// POUs/Functions/Pumps/FB_PTM_TurboDrive
(* This Function block provides basic turbo control for Leybold Turbo Drive 300, Turbo Drive 400 *)
(* TD20 Classic Via Remote X1 Connector 9-way PLC interface*)
FUNCTION_BLOCK FB_PTM_TurboDrive
VAR_IN_OUT
	
END_VAR
VAR_INPUT
	i_xExtILKOk : BOOL; // Connect to external interlock logic, TRUE if not used.
END_VAR
VAR_OUTPUT
{attribute 'pytmc' := '
    pv: 
	'}
	iq_stPtm	:	ST_LeyboldPTM;
END_VAR
VAR
	xRunOk	:	BOOL;
	tofRemoteDelay	:	TOF;
	
	
	(*IO*)
	i_xAtSpd AT%I*: BOOL; // Normaml operation when true
	i_xFaultNC AT%I*: BOOL; // Error Active when no Error is present
	q_RunDO AT%Q*: BOOL; // Start/Stop

END_VAR

(* Basic Turbo Control *)
(* This Function block provides basic turbo control for Leybold Turbo Drive 300, Turbo Drive 400 *)
(* TD20 Classic Via Remote X1 Connector 9-way PLC interface*)
(* M. Ghaly Jan. 2019 *)

(* Interlock Sum *)
iq_stPtm.xExtRunOk:= i_xExtILKOk;
xRunOk := iq_stPtm.xExtRunOk AND iq_stPtm.i_xNCError;

(* Basic pump supervisory section *)
IF xRunOk THEN
	iq_stPtm.q_RunDO := iq_stPTM.xRunSW;
ELSE
	iq_stPtm.xRunSW:=FALSE;
	iq_stPtm.q_RunDO:=FALSE;
END_IF

(*Pump States*)
IF (iq_stPtm.i_xFault) THEN
		iq_stPtm.eState := pumpFAULT;
		iq_stPtm.xRunSW:=FALSE;
		iq_stPtm.q_RunDO:=FALSE;
	ELSIF (iq_stPtm.q_RunDO) AND (iq_stPtm.i_xAtSpd) THEN
		iq_stPtm.eState := pumpRUNNING;
	ELSIF (iq_stPtm.q_RunDO) AND NOT (iq_stPtm.i_xAtSpd) THEN
		iq_stPtm.eState := pumpSTARTING; 
	ELSIF NOT (iq_stPtm.q_RunDO) THEN
		iq_stPtm.eState := pumpSTOPPED; 	
END_IF;
			

(*I/O soft mapping*)
ACT_IO();

ACTION ACT_IO:
(*Inputs*)
iq_stPtm.i_xAtSpd := i_xAtSpd;
iq_stPtm.i_xNCError := i_xFaultNC;
iq_stPtm.i_xFault := NOT i_xFaultNC;



(*Outputs*)
q_RunDO := iq_stPtm.q_RunDO;
END_ACTION

METHOD PUBLIC M_Run : BOOL
VAR_INPUT
	run:bool; // set to true to run, false to stop;
END_VAR

this^.iq_stPtm.xRunSW := run;
END_METHOD

END_FUNCTION_BLOCK

// POUs/Functions/Pumps/FB_PTM_TwisTorr
(* This function block does basic controls FOR the Agilent TwisTorr 304 FS with on board Controller.
 Turns off pump in the event of errors/ warnings. Provides interlocking interface.*)
FUNCTION_BLOCK FB_PTM_TwisTorr
VAR_INPUT
	i_xExtILKOk : BOOL; // Connect to external interlock logic, TRUE if not used.
	
END_VAR
VAR_OUTPUT
	{attribute 'pytmc' := ' pv: '}
	iq_stPtm	:	ST_PTM;
END_VAR
VAR
	xRunOk	:	BOOL;
	(*IO*)
	i_xAtSpd AT%I*: BOOL; // Normaml operation when true
	i_xFault AT%I*: BOOL; // Error // this open collector output signal is ON when a system fault condition is detected

	q_RunDO AT%Q*: BOOL; // Start/Stop

END_VAR


(* Interlock Sum *)
iq_stPtm.xExtRunOk:= i_xExtILKOk;
xRunOk := iq_stPtm.xExtRunOk AND NOT iq_stPtm.i_xFault;

(* Basic pump supervisory section *)
IF xRunOk THEN
	iq_stPtm.q_RunDO := iq_stPTM.xRunSW;
ELSE
	iq_stPtm.xRunSW:=FALSE;
	iq_stPtm.q_RunDO:=FALSE;
END_IF

(*Pump STATE*)
IF iq_stPtm.i_xFault THEN 
	iq_stPtm.eState := pumpFAULT;
ELSIF NOT iq_stPtm.q_RunDO AND NOT iq_stPTM.i_xFault THEN
	iq_stPtm.eState := pumpSTOPPED;
ELSIF NOT iq_stPtm.i_xAtSpd  AND iq_stPtm.q_RunDO THEN
	iq_stPtm.eState := pumpSTARTING;
ELSIF iq_stPtm.i_xAtSpd AND iq_stPtm.q_RunDO THEN
	iq_stPtm.eState := pumpRUNNING;
ELSE 
	iq_stPtm.eState := pumpFAULT;
END_IF

(*I/O soft mapping*)
ACT_IO();

ACTION ACT_IO:
(*Inputs*)
iq_stPtm.i_xAtSpd := i_xAtSpd;
iq_stPtm.i_xFault := i_xFault;


(*Outputs*)
q_RunDO := iq_stPtm.q_RunDO;
END_ACTION

METHOD PUBLIC M_Run : BOOL
VAR_INPUT
	run:bool; // set to true to run, false to stop;
END_VAR

this^.iq_stPtm.xRunSW := run;
END_METHOD

END_FUNCTION_BLOCK

// POUs/Functions/Pumps/FB_ScrollPump
(* This Function block provides basic  control for Scroll Pumps *)
(* Turn on scroll pump if the Turbo Vent Valve is closed. *)
(* Cannot turn off scroll pump if turb is running. delay scroll off 150s.*)  

FUNCTION_BLOCK FB_ScrollPump
VAR_IN_OUT

END_VAR
VAR_OUTPUT
	{attribute 'pytmc' := '
    pv:
	'}
	iq_stPFO	:	ST_RoughPump;
END_VAR
VAR_INPUT
	TurboIsON : BOOL;
	xExtIlk : BOOL;
END_VAR
VAR
	Tmr_TOF : TOF;
	tTimerDuration : Time:= T#150S;
	//Previous_RunSW : BOOL;
	// Digital Output to be linked
	q_xRunDo AT%Q*	:   BOOL; 
END_VAR

//Turn on scroll pump if the Turbo Vent Valve is closed. So you are not just
// pumping air and accomplishing nothing

// cannot turn off scroll pump if turb is running. delay scroll off 150s.  
iq_stPFO.xIlkOK := xExtIlk;// and NOT Tmr_TOF.Q;

Tmr_TOF(IN:=TurboIsON, PT := tTimerDuration);

IF iq_stPFO.xIlkOK THEN
	iq_stPFO.q_xRunDo := (Tmr_TOF.Q OR iq_stPFO.pv_xRunSW);
ELSE
	iq_stPFO.q_xRunDo := FALSE;
END_IF

iq_stPFO.pv_xRunSW := iq_stPFO.q_xRunDo;

(*State evaluation*)
IF NOT iq_stPFO.q_xRunDo THEN
	iq_stPFO.eState := pumpSTOPPED;	
ELSE
	iq_stPFO.eState := pumpRUNNING;
END_IF

(*soft io Mapping*)
IO();

ACTION IO:
q_xRunDo:= iq_stPFO.q_xRunDo;
END_ACTION

METHOD PUBLIC M_Run : BOOL
VAR_INPUT
	run:bool; // set to true to run, false to stop;
END_VAR

this^.iq_stPFO.pv_xRunSW := run;
END_METHOD

END_FUNCTION_BLOCK

// POUs/Functions/Valves/functions/F_RoughPumpInlet_ILK
(*
	Determine whether a pump attached to the inlet of a roughing pump is safe to open. 
	
	Return true, signaling it is safe to open when the roughing pump is confirmed to be working. 
*)

FUNCTION F_RoughPumpInlet_ILK : BOOL
VAR_INPUT
	ScrollPump	:	ST_RoughPump;
END_VAR
VAR
END_VAR


F_RoughPumpInlet_ILK := (ScrollPump.eState = pumpRUNNING); (* Confirm that the roughing pump is running before opening the valve *)

END_FUNCTION

// POUs/Functions/Valves/functions/F_TURBO_VRC_ILK
(* Close the vic if the roughing pump pirani loses its at-vac setpoint while the turbo is pumping *)
FUNCTION F_TURBO_VRC_ILK : BOOL
VAR_INPUT

	i_xHiVac 	: BOOL;
	i_xRunPTM	: BOOL;
	i_xFLVac	: BOOL;

END_VAR
VAR

	rHysterisis : REAL := 0;

	xInterlock: BOOL;
	rTolerance: REAL := 20;
END_VAR

(* Close the vic if the roughing pump pirani loses its at-vac setpoint while the turbo is pumping *)
F_TURBO_VRC_ILK := (NOT i_xHiVac AND NOT i_xRunPTM AND NOT i_xFLVac) OR
					(NOT i_xRunPTM AND i_xFLVac) OR
					(i_xRunPTM AND i_xFLVac);

END_FUNCTION

// POUs/Functions/Valves/functions/F_TurboGateValve_ILK
(* This Function Block evaluates the ILK condition of the Turbo Gate valve *)
(* The logic Protects the Turbo pump from inlet pressure above the SP*)

FUNCTION F_TurboGateValve_ILK : BOOL (* function return TRUE when ILK is OK*)
VAR_INPUT
	i_Turbo : ST_PTM; // Turbo Pump
	i_stISG : ST_VG; //Gauge measuring inlet Pressure e.g Pirani
END_VAR
VAR
END_VAR

(* This Function Block evaluates the ILK condition of the Turbo Gate valve *)
(* The logic Protects the Turbo pump from inlet pressure above the SP*)
F_TurboGateValve_ILK := (NOT (i_Turbo.eState = pumpSTOPPED) AND NOT (i_Turbo.eState = pumpFAULT))
						AND (i_stISG.xPRESS_OK AND i_stISG.rPRESS < i_Turbo.rInletPressureSP);

END_FUNCTION

// POUs/Functions/Valves/functions/F_TurboGateValve_Protection_ILK
(* This Function Block evaluates the ILK condition of the Turbo Gate valve *)
(* The logic Protects the Turbo pump from inlet pressure above the SP*)
(* And Protects the Turbo pump from backing pressure above the SP*)
(* And Protects the Turbo pump in the case of backing pump not running*)

FUNCTION F_TurboGateValve_Protection_ILK : BOOL (* function return TRUE when ILK is OK*)
VAR_INPUT
	i_Turbo : ST_PTM; // Turbo Pump
	i_stISG : ST_VG; //Gauge measuring inlet Pressure e.g Pirani
	i_stBSG : ST_VG; //Gauge measuring backing Pressure e.g Pirani
	ScrollPump	:	ST_RoughPump; // Roughing pump
END_VAR
VAR
END_VAR

(* This Function Block evaluates the ILK condition of the Turbo Gate valve *)
(* The logic Protects the Turbo pump from inlet pressure above the SP*)
F_TurboGateValve_Protection_ILK := (NOT (i_Turbo.eState = pumpSTOPPED) AND NOT (i_Turbo.eState = pumpFAULT))
						AND (i_stISG.xPRESS_OK AND i_stISG.rPRESS < i_Turbo.rInletPressureSP)
						AND (i_stBSG.xPRESS_OK AND i_stBSG.rPRESS < i_Turbo.rBackingPressureSP)
						AND (ScrollPump.eState = pumpRUNNING);

END_FUNCTION

// POUs/Functions/Valves/functions/F_VALVE_REL_ILK
(* OK, this is going to be a general-use function that will return whether the ratio of the pressures given is less than x orders of magnitude.
True iff 10^(-x) < a/b < 10^x.  Simple, right?  Just make sure it gets a positive order of magnitude and the pressures aren't 0. ~Scott *)   

FUNCTION F_VALVE_REL_ILK : BOOL
VAR_INPUT
	i_stUSG	:	ST_VG; // Upstream Gague
	i_stDSG	:	ST_VG; // Downstream Gague
	//Orders of magnitude allowed between up/downstream pressures for valve to open. Must be real positive integer.
	i_iOrdersMagnitude: INT;
END_VAR
VAR
	rPressRatio : REAL;
	rMaxRatioAllowed	:	LREAL := EXPT(10,i_iOrdersMagnitude);
	rMinRatioAllowed	:	LREAL := EXPT(10,(-i_iOrdersMagnitude));
END_VAR

(* S. Stubbs 11/2015 *)

(* OK, this is going to be a general-use function that will return whether the ratio of the pressures given is less than x orders of magnitude.
True iff 10^(-x) < a/b < 10^x.  Simple, right?  Just make sure it gets a positive order of magnitude and the pressures aren't 0. ~Scott *)   

(* Find ratio *)

IF i_stDSG.rPRESS <> 0 THEN
	rPressRatio := i_stUSG.rPRESS / i_stDSG.rPRESS;

	F_VALVE_REL_ILK := rPressRatio < rMaxRatioAllowed AND rMinRatioAllowed < rPressRatio;
ELSE
	F_VALVE_REL_ILK := FALSE;
END_IF

END_FUNCTION

// POUs/Functions/Valves/functions/F_VRC_DIODE_ILK
(* The principle is simple, a VRC should never open when B side pressure is greater than 
the A side pressure. *)

FUNCTION F_VRC_DIODE_ILK : BOOL
VAR_INPUT

	i_stPGA : ST_VG; // A side pressure gauge
	i_stPGB	: ST_VG; // B side pressure gauge

END_VAR
VAR

	rHysterisis : REAL := 0;

	xInterlock: BOOL;
	rTolerance: REAL := 20;
END_VAR

(* The principle is simple, a VRC should never open when B side pressure is greater than the A side pressure. *)
rTolerance := 20;
F_VRC_DIODE_ILK := ((i_stPGA.rPRESS + rTolerance >= i_stPGB.rPRESS + rHysterisis) OR i_stPGA.xBAKEOUT) AND i_stPGA.xPRESS_OK AND i_stPGB.xPRESS_OK;

(* OK it gets a bit more complicated with hysterisis,

Now, if the F_VIC_DIODE_ILK is FALSE then some hysterisis is added to the B side. But if it's OK then we just stick with making sure that the A side is greater than the B side

*)
(*
IF NOT F_VIC_DIODE_ILK THEN
Hysterisis := 40;
ELSE
Hysterisis := 0;
END_IF
*)

END_FUNCTION

// POUs/Functions/Valves/Interfaces/FB_TVGC_ADS
(* This function block is created for interface devices between different PLC*)
(* Not all the fields in the original structure is required, just few signals *)
(*Use with FB_ADS_WATCHDOG on remotePLC*)
FUNCTION_BLOCK FB_TVGC_ADS
VAR_INPUT
	sNetId : String; //NetID of the Destination PLC controller
	nPort : int; // port number
	sVarName : string;// the variable name of the (device) declared function block.
	iWatchdog:UDINT;//The watchdog variable name written to by the remote plc
END_VAR
VAR_OUTPUT
	{attribute 'pytmc' := 'pv: '}
	VGC:ST_VGC;
	bError:BOOL;
END_VAR
VAR
	fb_CheckWatchdog: FB_CheckWatchdog;
	fb_Read_VGC: FB_ReadAdsSymByName;
	ftReset: F_TRIG;
	xFirstPass: bool:= true;
END_VAR

ftReset(CLK:= fb_Read_VGC.bBusy OR xFirstPass);
xFirstPass:=false;
(*calling ADS read function*)
fb_Read_VGC(
	bRead:= ftReset.Q, 
	sNetId:= sNetId, 
	nPort:= nPort, 
	sVarName:= CONCAT(sVarName,'.iq_stValve'), 
	nDestAddr:= ADR(VGC), 
	nLen:= SIZEOF(VGC), 
	tTimeout:= , 
	eComMode:= eAdsComModeFastCom, 
	bBusy=> , 
	bError=> , 
	nErrorId=> );
	

(*Error*)
fb_CheckWatchdog(
	bEnable:= TRUE, 
	tWatchdogTime:= T#100ms, 
	nCnt:= iWatchdog , 
	bWatchdog=> , 
	nLastCnt=> );
bError:= fb_Read_VGC.bError OR fb_CheckWatchdog.bWatchdog;

END_FUNCTION_BLOCK

// POUs/Functions/Valves/Interfaces/FB_Valve_Interface
(* This function block is created for interface devices between different PLC*)
(* Not all the fields in the original structure is required, just few signals *)
(* They have to be linked to the custom created variables on the EL6692/5 primary side*)

FUNCTION_BLOCK FB_Valve_Interface
VAR_INPUT
END_VAR
VAR_OUTPUT
	{attribute 'pytmc' := 'pv: '}
	VGC:ST_VGC;
END_VAR
VAR
	i_xOpnLS AT%I*	: BOOL;
	i_xClsLS AT%I*	: BOOL;
END_VAR

(* This function block is created for interface devices between different PLC*)
(* Not all the fields in the original structure is required, just few signals *)
(* They have to be linked to the custom created variables on the EL6692/5 primary side*)


VGC.i_xClsLS := i_xClsLS;
VGC.i_xOpnLS := i_xOpnLS;

END_FUNCTION_BLOCK

// POUs/Functions/Valves/Interfaces/FB_VFS_Interface
(*Used as soft IO mapping to create a psuedo valve to communicate over two task on the same PLC.*) 
(*for FAST shutter control*)
FUNCTION_BLOCK FB_VFS_Interface
VAR_INPUT
	IG : ST_VG; // The Cold Cathode Data Structure
	{attribute 'pytmc' := '
    pv: FF_Reset
	'}
    i_xFFReset: BOOL;
END_VAR
VAR_IN_OUT
	io_fbFFHWO    :    FB_HardwareFFOutput;
END_VAR
VAR
	// PMPS
	fbFF    :    FB_FastFault :=(
        i_DevName := 'VGC',
        i_Desc := 'Fault occurs when fast sensor trips or the valve is not in open state',
        i_TypeCode := 16#1010);

	(*outputs*)
	q_xPRESS_OK AT%Q*: BOOL;
	{attribute 'pytmc' := '
	pv: CLS_SW; 
	io: io ;
	'}
	q_xCLS_SW AT%Q*:BOOL; (*external open signal e.g epics*)
	{attribute 'pytmc' := '
	pv: FAULT_RESET; 
	io: io ;
	'}
	q_xVAC_FAULT_Reset AT%Q*: BOOL; (*Valve Vacuum OK, is set to False when there is Vacuum Fault*)

	
	(*inputs*)
	{attribute 'pytmc' := '
	pv: TRIG; 
	field: ZNAM TRIG_OFF; 
	field: ONAM TRIG_ON;
	io: io ;
	'}
	i_xTrigger AT %I* : BOOL;
	{attribute 'pytmc' := '
	pv: OPEN; 
	field: ZNAM NOT OPEN; 
	field: ONAM OPEN;
	io: io ;
	'}
	i_xVFS_Open AT %I* : BOOL;
	{attribute 'pytmc' := '
	pv: CLS; 
	field: ZNAM NOT CLOSED; 
	field: ONAM CLOSE;
	io: io ;
	'}
	i_xVFS_Closed AT %I* : BOOL;
	{attribute 'pytmc' := '
	pv: FAULT_OK; 
	field: ZNAM FAULT ; 
	field: ONAM FAULT OK;
	io: io ;
	'}
	i_xVAC_FAULT_OK AT%I*: BOOL; (*Valve Vacuum OK, is set to False when there is Vacuum Fault*)
	{attribute 'pytmc' := '
	pv: FFO_OK; 
	field: ZNAM FAULT ; 
	field: ONAM FAULT OK;
	io: io ;
	'}
	i_xMPS_OK AT%I*: BOOL;(*MPS Fault OK, is set when the Valve is Open and there is no trigger*)
END_VAR

(*soft IO Mapping*)

q_xPRESS_OK := IG.xPRESS_OK;

(*FAST FAULT*)
fbFF(i_xOK := i_xMPS_OK,
    i_xReset := i_xFFReset,
    io_fbFFHWO := io_fbFFHWO);

END_FUNCTION_BLOCK

// POUs/Functions/Valves/Interfaces/ITF_Valve
INTERFACE ITF_Valve

END_INTERFACE

// POUs/Functions/Valves/FB_Kashiyama_VRC
(* Main Kashiyama gate valve permit to be open when:
		1. pump is NORMAL operating status, and
	    2. chamber pressure is below HighSP or pump is at LowSpeed state.
	it will close if chamber pressure is below than lowSP for 180s.	
*)
FUNCTION_BLOCK FB_Kashiyama_VRC
VAR_IN_OUT
	
END_VAR
VAR_OUTPUT
	{attribute 'pytmc' := ' pv:'}
	q_stValve : ST_VRC;
END_VAR
VAR_INPUT
	Pump : ST_KashiyamaDryPump;//Kashyiama pump
	i_xExtILK_OK : BOOL; //Connect to Interlock logic condition(e.g F_TURBO_VRC_ILK Function), otherwise, Set to True if the valve is not interlocked
	Gauge : ST_VG;// Pressure Gauge	
	i_xOverrideMode : BOOL;
END_VAR
VAR
	At_HiVac : BOOL;
	tmrTP : TP;
	tmrPT: TIME := T#180S;
	v1: BOOL;
	tonOvrd	:	TON;
	tonDelOK : TON;
	rtOK	:	R_TRIG;
	
	(*IO*)
	i_xOpnLS	AT%I*: BOOL;
	i_xClsLS	AT%I*: BOOL;
	q_xOPN_DO	AT%Q*: BOOL;
	
END_VAR

(* Main Kashiyama gate valve permit to be open when:
		1. pump is NORMAL operating status, and
	    2. chamber pressure is below HighSP or pump is at LowSpeed state.
	it will close if chamber pressure is below than lowSP for 60s.	
*)
(* 
      For main Kayshiyama pump's gate valve:
		Pump LowSP is MU100 base pressure (20 mTorr) 
		Pump HighSP is 600 Torr;
	  Second Kayshiyama pump allow Gas Attenuator operating at higher pressure, 
      it's gate valve is to be open when Gas Attenuator chamber pressure is above lowSP.  
*)


///Check valve postion
IF NOT q_stValve.i_xClsLS AND q_stValve.i_xOpnLS THEN 
	q_stValve.eState:=OPEN;
ELSIF q_stValve.i_xClsLS AND NOT q_stValve.i_xOpnLS THEN 
	q_stValve.eState:=CLOSED;
ELSIF NOT q_stValve.i_xClsLS AND NOT q_stValve.i_xOpnLS THEN 
	q_stValve.eState:=MOVING;
ELSE
	q_stValve.eState:=INVALID;
END_IF

//valve open interlock
q_stValve.xOPN_OK := Pump.i_xIsRun AND Pump.RdyTmr <= 0.0 AND (Gauge.rPRESS < Pump.HighSP OR Pump.q_xLspdDo) AND i_xExtILK_OK;
 

(* Override logic *)
(* Goal: give ability to override, but do so in a way that people won't forget it.
Solution: Override only after ten seconds of override, protect against blips,
when the valve permission goes true for more than ten seconds consistently, remove override
*)

tonDelOK(IN:=q_stValve.xOPN_OK, PT:=T#10S);
rtOK(CLK:=tonDelOK.Q);
IF rtOK.Q THEN q_stValve.pv_xOvrdOpn :=FALSE; END_IF

//Override timer
tonOvrd(IN:=q_stValve.pv_xOvrdOpn, PT:=T#10S);


(* Here's where the valve closes *)
IF NOT q_stValve.xOPN_OK AND NOT tonOvrd.Q THEN
q_stValve.pv_xOPN_SW := FALSE;
END_IF

At_HiVac := Gauge.xPRESS_OK AND Gauge.rPRESS < Pump.LowSP;
tmrTP (IN := At_HiVac AND q_stValve.q_xOPN_DO , PT := tmrPT);

IF At_HiVac AND q_stValve.q_xOPN_DO AND NOT tmrTP.Q THEN
	q_stValve.pv_xOPN_SW := FALSE ;
END_IF

(* Here's where the valve opens *)
q_stValve.q_xOPN_DO := (q_stValve.pv_xOPN_SW AND q_stValve.xOPN_OK) OR (tonOvrd.Q AND i_xOverrideMode); 

(*Soft IO Mapping*)
ACT_IO();

ACTION ACT_IO:
(*inputs*)
q_stValve.i_xOpnLS := 	i_xOpnLS;
q_stValve.i_xClsLS:=	i_xClsLS;
(*outputs*)
q_xOPN_DO:= q_stValve.q_xOPN_DO;
END_ACTION

END_FUNCTION_BLOCK

// POUs/Functions/Valves/FB_MKS248
(* MKS248 valve using MKS1249 Drive Module *)
FUNCTION_BLOCK FB_MKS248
VAR_INPUT
	i_xExtIlkOK	:	BOOL; //External Interlock, SET to TRUE if not used
	i_rReqPos	:	REAL; //Requested position
END_VAR
VAR_OUTPUT
	{attribute 'pytmc' := 'pv:'}
	iq_stVFN	:	ST_VCN; //Needle valve structure
END_VAR
VAR CONSTANT
	rOpenVoltage	:	REAL := 9.8; 
	rCloseVoltage	:	REAL := 0;	
END_VAR
VAR
	// Requested voltage
	rReqVoltage: REAL := 0;
	(*IO*)
	q_iRawPosition AT%Q* :INT;
END_VAR

(* MKS248 valve using MKS1249 Drive Module *)


// Interlocking
iq_stVFN.xIlkOK := i_xExtIlkOK;
(*Checking which Control mode is selected*)
IF iq_stVFN.xIlkOK THEN
	IF iq_stVFN.eValveControl = OpenValve THEN
		iq_stVFN.rReqPosition := iq_stVFN.rUpperLimit;(*Percentage*)// iq_stVCN.rUpperLimit;
	ELSIF iq_stVFN.eValveControl = CloseValve THEN
		iq_stVFN.rReqPosition := 0; (*Percentage*)
	ELSIF iq_stVFN.eValveControl = ManualControl THEN
		iq_stVFN.rReqPosition := LIMIT(0, iq_stVFN.rReqPosition, iq_stVFN.rUpperLimit);
	ELSIF iq_stVFN.eValveControl = PressureControl THEN
		iq_stVFN.rReqPosition := LIMIT(0, i_rReqPos, iq_stVFN.rUpperLimit); 
	END_IF
ELSE
	iq_stVFN.rReqPosition := 0;
	iq_stVFN.eValveControl := CloseValve;
END_IF

// Requested Voltage calculation
rReqVoltage := iq_stVFN.rReqPosition * (rOpenVoltage-rCloseVoltage)/100 + rCloseVoltage;
rReqVoltage := LIMIT(rCloseVoltage, rReqVoltage, rOpenVoltage); //The requested voltage should remain within this range
//Raw position calc
iq_stVFN.q_iRawPosition := REAL_TO_INT( 32767/10 * rReqVoltage);	
(*IO Mapping*)
ACT_IO();

ACTION ACT_IO:
(*outputs*)
q_iRawPosition := iq_stVFN.q_iRawPosition;
END_ACTION

END_FUNCTION_BLOCK

// POUs/Functions/Valves/FB_TurbVentvalve_NO
(* This function block impelemets Interlock for Agilent Turbo Vent Valve Normally Open*)
FUNCTION_BLOCK FB_TurbVentvalve_NO
VAR_OUTPUT
	{attribute 'pytmc' :=' pv:'}
	q_stValve : ST_VCC_NO;
END_VAR
VAR_INPUT
	i_stPTM	: ST_AgilentPTM; //Agilent Turbo Pump
END_VAR
VAR
	tofTmr 		: 	TOF;
	
	(*Output*)
	q_xCLS_DO AT%Q* : BOOL;
END_VAR

(*If the turbo is on, you cannot open the valve. In order to open the valve, you have to allow the turbopump
 to have already been turned off for 2 minutes and you have to press the open button on the vent valve

If the code looks confusing please use a truth table to verify*)

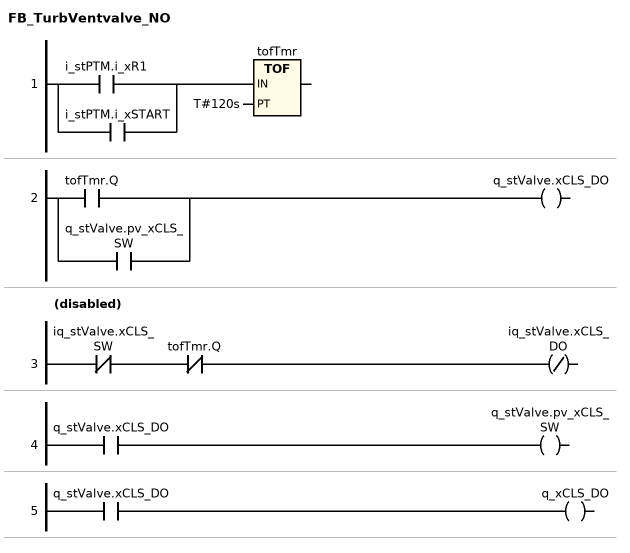
// NETWORK 1
tofTmr(IN := i_stPTM.i_xR1 OR i_stPTM.i_xSTART, PT := T#120s); // TOF

// NETWORK 2
q_stValve.xCLS_DO := tofTmr.Q OR q_stValve.pv_xCLS_SW;

// NETWORK 3 (disabled)
// iq_stValve.xCLS_DO := NOT (NOT iq_stValve.xCLS_SW AND NOT tofTmr.Q);

// NETWORK 4
q_stValve.pv_xCLS_SW := q_stValve.xCLS_DO;

// NETWORK 5
q_xCLS_DO := q_stValve.xCLS_DO;

ACTION ACT_IO:
(*outputs*)
q_xCLS_DO:= q_stValve.xCLS_DO;
END_ACTION

METHOD M_Close : BOOL
VAR_INPUT
		close:BOOL; //True to CLose, False to OPEN
END_VAR
This^.q_stValve.pv_xCLS_SW :=Close;
END_METHOD

END_FUNCTION_BLOCK

// POUs/Functions/Valves/FB_VCC
(* THE FB_VCC FUNCTION BLOCK IS DEPRECATED. USE FB_VVC INSTEAD. *)
(* This Function Block Implements Basic Functionality for Vent Valves VVC *)
(* Note Interlock Logic is External *)
FUNCTION_BLOCK FB_VCC
VAR_IN_OUT

END_VAR
VAR_INPUT
	i_xExtILK_OK:BOOL; (*Other External Interlock, Set to True when no external interlock is required*)
	i_xOverrideMode : BOOL; (*To be linked to global override bit. This Overrides Vacuum logic only*)
END_VAR
VAR_OUTPUT
	{attribute 'pytmc' := '
    pv:
	'}
	iq_stValve : ST_VVC;
END_VAR
VAR

	tonOvrd	:	TON;
	tonDelOK : TON;
	rtOK	:	R_TRIG;

	(*IO*)
	q_xOPN_DO	AT%Q*: BOOL;

END_VAR


iq_stValve.xOPN_OK := i_xExtILK_OK;

IF NOT iq_stValve.xOPN_OK THEN
iq_stValve.pv_xOPN_SW := FALSE;
END_IF

(* Override logic *)
(* Goal: give ability to override, but do so in a way that people won't forget it.
Solution: Override only after ten seconds of override, protect against blips,
when the valve permission goes true for more than ten seconds consistently, remove override
*)

tonDelOK(IN:=iq_stValve.xOPN_OK, PT:=T#10S);
rtOK(CLK:=tonDelOK.Q);
IF rtOK.Q THEN iq_stValve.xOvrdOpn :=FALSE; END_IF

//Override timer
tonOvrd(IN:=iq_stValve.xOvrdOpn, PT:=T#10S);

(* Here's where the valve opens *)
iq_stValve.q_xOPN_DO := (iq_stValve.pv_xOPN_SW AND iq_stValve.xOPN_OK) OR (tonOvrd.Q AND i_xOverrideMode);

(*IO Mapping*)
ACT_IO();

ACTION ACT_IO:
(*inputs*)
iq_stValve.xOverrideMode := i_xOverrideMode;
(*outputs*)
q_xOPN_DO:= iq_stValve.q_xOPN_DO;
END_ACTION

METHOD PUBLIC M_IsClosed : BOOL
VAR_INPUT
END_VAR
M_IsClosed := NOT This^.q_xOPN_DO;
END_METHOD

METHOD PUBLIC M_IsOpen : BOOL
VAR_INPUT
END_VAR
M_IsOpen := This^.q_xOPN_DO;
END_METHOD

// Use this Methode to Open or close the valve by setting the OPN_SW to the input value.
METHOD PUBLIC M_Set_OPN_SW : BOOL
VAR_INPUT
		value:BOOL;  //True to SET, False to RESET
END_VAR
This^.iq_stValve.pv_xOPN_SW := value;
END_METHOD

END_FUNCTION_BLOCK

// POUs/Functions/Valves/FB_VVC
(* This Function Block Implements Basic Functionality for Vent Valves VVC.

	This function block is also intended for the general use case of solenoid driven (non-variable) valves that lack status readbacks or position indicators. 
*)
(* Note Interlock Logic is External *)
FUNCTION_BLOCK FB_VVC
VAR_IN_OUT

END_VAR
VAR_INPUT
	i_xExtILK_OK:BOOL; (*Other External Interlock, Set to True when no external interlock is required*)
	i_xOverrideMode : BOOL; (*To be linked to global override bit. This Overrides Vacuum logic only*)
END_VAR
VAR_OUTPUT
	{attribute 'pytmc' := '
    pv:
	'}
	iq_stValve : ST_VVC;
END_VAR
VAR

	tonOvrd	:	TON;
	tonDelOK : TON;
	rtOK	:	R_TRIG;

	(*IO*)
	q_xOPN_DO	AT%Q*: BOOL;

END_VAR


iq_stValve.xOPN_OK := i_xExtILK_OK;

IF NOT iq_stValve.xOPN_OK THEN
iq_stValve.pv_xOPN_SW := FALSE;
END_IF

(* Override logic *)
(* Goal: give ability to override, but do so in a way that people won't forget it.
Solution: Override only after ten seconds of override, protect against blips,
when the valve permission goes true for more than ten seconds consistently, remove override
*)

tonDelOK(IN:=iq_stValve.xOPN_OK, PT:=T#10S);
rtOK(CLK:=tonDelOK.Q);
IF rtOK.Q THEN iq_stValve.xOvrdOpn :=FALSE; END_IF

//Override timer
tonOvrd(IN:=iq_stValve.xOvrdOpn, PT:=T#10S);

(* Here's where the valve opens *)
iq_stValve.q_xOPN_DO := (iq_stValve.pv_xOPN_SW AND iq_stValve.xOPN_OK) OR (tonOvrd.Q AND i_xOverrideMode);

(*IO Mapping*)
ACT_IO();

ACTION ACT_IO:
(*inputs*)
iq_stValve.xOverrideMode := i_xOverrideMode;
(*outputs*)
q_xOPN_DO:= iq_stValve.q_xOPN_DO;
END_ACTION

// Method Returns True if the Valve is closed, i.e. the open digital output is not active
METHOD PUBLIC M_IsClosed : BOOL
VAR_INPUT
END_VAR
M_IsClosed := NOT This^.q_xOPN_DO;
END_METHOD

// Method Returns True if the Valve is open, i.e. the open digital output is active
METHOD PUBLIC M_IsOpen : BOOL
VAR_INPUT
END_VAR
M_IsOpen := This^.q_xOPN_DO;
END_METHOD

METHOD PUBLIC M_Open : BOOL
VAR_INPUT
	open: bool; //Set to true to open the valvue, false to close
END_VAR
This^.iq_stValve.pv_xOPN_SW := open;
END_METHOD

// Use this Methode to Open or close the valve by setting the OPN_SW to the input value.
METHOD PUBLIC M_Set_OPN_SW : BOOL
VAR_INPUT
	value:BOOL; //True to SET, False to RESET
END_VAR
This^.iq_stValve.pv_xOPN_SW := value;
END_METHOD

END_FUNCTION_BLOCK

// POUs/Functions/Valves/FB_VCC_NO
(* This Function Block Implements Basic Functionality for NO Vent Valves VVC *)
(* Note Interlock Logic is External *)
FUNCTION_BLOCK FB_VCC_NO
VAR_IN_OUT
	{attribute 'pytmc' := 'pv:'}
	iq_stValve : ST_VCC_NO;

END_VAR
VAR_INPUT
	i_xExtILK_OK:BOOL; (*Other External Interlock, Set to True when no external interlock is required*)
	i_xOverrideMode : BOOL; (*To be linked to global override bit. This Overrides Vacuum logic only, EPS, MPS and PMPS are still enforces*)

END_VAR
VAR_OUTPUT
END_VAR
VAR

	tonOvrd	:	TON;
	tonDelOK : TON;
	rtOK	:	R_TRIG;
	(*IO*)
	xCLS_DO	AT%Q*: BOOL;

END_VAR


IF NOT iq_stValve.xCLS_OK THEN
iq_stValve.pv_xCLS_SW := FALSE;
END_IF

(* Override logic *)
(* Goal: give ability to override, but do so in a way that people won't forget it.
Solution: Override only after ten seconds of override, protect against blips,
when the valve permission goes true for more than ten seconds consistently, remove override
*)

tonDelOK(IN:=iq_stValve.xCLS_OK, PT:=T#10S);
rtOK(CLK:=tonDelOK.Q);
IF rtOK.Q THEN iq_stValve.pv_xOvrdCls :=FALSE; END_IF

//Override timer
tonOvrd(IN:=iq_stValve.pv_xOvrdCls, PT:=T#10S);

(* Here's where the valve is closed *)
iq_stValve.xCLS_DO := (iq_stValve.pv_xCLS_SW AND iq_stValve.xCLS_OK) OR (tonOvrd.Q AND i_xOverrideMode);

ACTION ACT_IO:
(*inputs*)
iq_stValve.xOverrideMode := i_xOverrideMode;
(*outputs*)
xCLS_DO:= iq_stValve.xCLS_DO;
END_ACTION

METHOD M_Close : BOOL
VAR_INPUT
		close:BOOL; //True to CLose, False to OPEN
END_VAR
This^.iq_stValve.pv_xCLS_SW :=Close;
END_METHOD

END_FUNCTION_BLOCK

// POUs/Functions/Valves/FB_VCN
(* This function implements the Basic functions for the Pfeiffer EVR 116 needle valve*)
FUNCTION_BLOCK FB_VCN
VAR_INPUT
	i_xExtIlkOK	:	BOOL; //External Interlock, SET to TRUE if not used
	i_ReqPos	:	REAL; //Requested position

END_VAR
VAR_OUTPUT
	{attribute 'pytmc' := '
    pv:
	'}
	iq_stVCN	:	ST_VCN; //Needle valve structure
END_VAR
VAR_IN_OUT
	
END_VAR

VAR CONSTANT
	rOpenVoltage	:	REAL := 9.1; // From the EVR 116 manual, A Voltage of 9V it is completely Open
	rCloseVoltage	:	REAL := 0.4;// a voltage <0.5 V the valve is closed	
END_VAR
VAR
	// Requested voltage
	rReqVoltage: REAL := 0;
	//iResolution: INT :=16;
	// 
	(*IO*)
	q_iRawPosition AT%Q* :INT;

END_VAR

(* Needle valve control FB
A. Wallace 2016-7-21

This FB should be used as a low level control block.

It provides:

Valve position ceiling
Interlock
Scaling

It is not intended for:
Closed-loop control

It could be used for:
Valve position/flow linearization

Note: Raw position calc is based on 0.5 to 9V span, 32767 bits
*)

// Interlocking
iq_stVCN.xIlkOK := i_xExtIlkOK;
(*Checking which Control mode is selected*)
IF iq_stVCN.xIlkOK THEN
	IF iq_stVCN.eValveControl = OpenValve THEN
		iq_stVCN.rReqPosition := iq_stVCN.rUpperLimit;(*Percentage*)// iq_stVCN.rUpperLimit;
	ELSIF iq_stVCN.eValveControl = CloseValve THEN
		iq_stVCN.rReqPosition := 0; (*Percentage*)
	ELSIF (iq_stVCN.eValveControl = ManualControl) (*AND (iq_stVCN.xOPN_SW)*) THEN
		iq_stVCN.rReqPosition := LIMIT(0, iq_stVCN.rReqPosition, iq_stVCN.rUpperLimit);
	ELSIF iq_stVCN.eValveControl = PressureControl THEN
		iq_stVCN.rReqPosition := LIMIT(0, i_ReqPos, iq_stVCN.rUpperLimit); 
	END_IF
ELSE
	iq_stVCN.rReqPosition := 0;
	iq_stVCN.eValveControl := CloseValve;
END_IF

// Requested Voltage calculation
rReqVoltage := iq_stVCN.rReqPosition * (rOpenVoltage-rCloseVoltage)/100 + rCloseVoltage;
rReqVoltage := LIMIT(rCloseVoltage, rReqVoltage, rOpenVoltage); //The requested voltage should remain within this range
//Raw position calc
iq_stvcn.q_iRawPosition := REAL_TO_INT( 32767/10 * rReqVoltage);	

(*SOft IO Mapping*)
ACT_IO();

ACTION ACT_IO:
(*outputs*)
q_iRawPosition := iq_stVCN.q_iRawPosition;
(*inputs*)
iq_stVCN.i_iPosition := iq_stvcn.q_iRawPosition;
END_ACTION

METHOD M_ValveControl : BOOL
VAR_INPUT
	state:E_VCN; // Close, Open, Pressure, Manual
END_VAR
iq_stVCN.eValveControl := state;
END_METHOD

END_FUNCTION_BLOCK

// POUs/Functions/Valves/FB_VFS
FUNCTION_BLOCK FB_VFS
(* This function block implements basic functionality for Fast Shutter/Valves*)
(* Create a separate virtual PLC for the fast shutter logic, and tie/map this task to the FAST I/O portion of the ethercat bus,
 so we can scan these I/Os faster than the rest of the vacuum I/Os.
The Fast shutter was tested with PLC task Cycle Base Time 50us with cycle time 0.050ms.
*)
VAR_IN_OUT
	
END_VAR
VAR_INPUT

	i_xPMPS_OK:	BOOL	; (*External MPS interlock, Set to TRUE when no PMPS interlock is required*)
	i_xExt_OK: BOOL; (*Other External Interlock, Set to True when no external interlock is required*)
	i_xOverrideMode : BOOL; (*To be linked to global override bit. This Overrides Vacuum logic only, EPS, MPS and PMPS are still enforces*)
	

END_VAR
VAR_OUTPUT

	iq_stValve : ST_VGC; (* All valve data and states will be in this struct*)
	
	
END_VAR	
VAR_IN_OUT
	
	
END_VAR
VAR
	
	
	rDiffPressAllowed	:	REAL := 22.5; // Torr, Default value comes from Vat Valve Manual
	rDiffPress : REAL;
	set : BOOL;
    reset: BOOL;
	  
	xFirstPass	:	BOOL;
	fbFSInit		:	R_TRIG;
	
	tonDelOK : TON;
	rtOK	:	R_TRIG;
	tonOvrd	:	TON;
	
	tDelOK	:	TIME := T#60S;
	tOvrd	:	TIME := T#10s;
	
	xClose: BOOL;
	xOpen: BOOL;
	CloseTimer: TON;
	TimDur: TIME := T#20MS;
	OpenTimer: TON;
	OpenTimDur: TIME := T#10S;
	
	(* Timeouts*)
	tTimeOutDuration: TIME:= T#0.5S;
	tOPNtimeout: TON;
	tCLStimeout:TON;
	

	i_xCLS_SW AT%I*:BOOL; (*external open signal e.g epics*)
	(*IO*)
	i_xOpnLS	AT%I*: BOOL;
	i_xClsLS	AT%I*: BOOL;
	q_xClose_A	AT%Q*: BOOL;
	q_xClose_B	AT%Q*: BOOL;
	q_xClose_C	AT%Q*: BOOL;
	q_xOPN_DO	AT%Q*: BOOL;
	i_xTrigger	AT%I*: BOOL; // Could be Up to 4
	
	// Interface
	i_xPress_OK AT%I*:BOOL; (*To be linked to the Fast sensor structure signal IG.xPRESS_OK, to make sure that the device is connected*)
	i_xResetFault	AT%I*: BOOL;(*FFO iReset*)
	q_xTrigger	AT%Q*: BOOL; (*Interface*)
	q_xVFS_Open AT%Q*: BOOL; (*Interface*)
	q_xVFS_Closed AT%Q*: BOOL; (*Interface*)
	q_xVAC_FAULT_OK AT%Q*: BOOL; (*Valve Vacuum OK, is set to False when there is Vacuum Fault*)
	q_xMPS_OK	 AT%Q*:	BOOL; (*MPS Fault OK, is set when the Valve is Open and there is no trigger*)
	
	
END_VAR



(* Fast Shutter/Valve Function Block*)
(* M.Ghaly Feb 2019*)

(* Fast Shutters do not function as complete isolation valves, but are intended to rapidly limit conductance 
between vacuum regions.  They should be installed in conjunction with isolation gate valves.  The conductance 
of the fast shutter in the closed state may be sufficiently low as to create an isolated vacuum region.  
Thus, at least a pirani gauge, that can measure a pressure down to 1x10-4 Torr, needs to be installed between
the shutter and the isolation gate valve.
In the case where a gauge is not installed, the neigboring gate Valves should not be opened unless the shutter 
is Open. 
*)
(* Soft IO Mapping*)
IO();

///Check valve postion
IF iq_stValve.i_xClsLS AND  iq_stValve.i_xOpnLS THEN
	iq_stValve.eState:=INVALID;
ELSIF NOT iq_stValve.i_xClsLS AND iq_stValve.i_xOpnLS AND iq_stValve.q_xOPN_DO THEN 
	iq_stValve.eState:=OPEN;
ELSIF iq_stValve.i_xClsLS AND NOT iq_stValve.i_xOpnLS AND NOT iq_stValve.q_xOPN_DO THEN 
	iq_stValve.eState:=CLOSED;
ELSIF NOT iq_stValve.i_xClsLS AND NOT iq_stValve.i_xOpnLS THEN 
	iq_stValve.eState:=MOVING;
ELSE
	iq_stValve.eState:=INVALID;
END_IF


(* Here's where the valve opens *)
//iq_stValve.q_xOPN_DO := (NOT(i_xCLS_SW) AND iq_stValve.xOPN_OK AND NOT i_xOpnLS) OR (tonOvrd.Q AND i_xOverrideMode);


(* Input Trigger to close the Fast Shutter*)
(* Neighboring Valves Should also be triggered to Close*)
IF (i_xTrigger) OR NOT (i_xPress_OK) OR NOT (i_xExt_OK)  OR i_xCLS_SW  THEN 
	xClose:= TRUE;
	iq_stValve.pv_xOPN_SW := FALSE;
	q_xVAC_FAULT_OK:= FALSE;
	IF (NOT i_xCLS_SW) THEN iq_stValve.xERR_ExtFault := TRUE; END_IF;
	i_xCLS_SW := TRUE;
	iq_stValve.q_xOPN_DO := FALSE;
	iq_stValve.pv_xOPN_SW :=FALSE;
	xOpen:=FALSE;
ELSIF ((iq_stValve.pv_xOPN_SW) AND iq_stValve.xOPN_OK ) OR (tonOvrd.Q AND i_xOverrideMode) THEN
	iq_stValve.q_xOPN_DO := TRUE;
	xOpen:=TRUE;
END_IF
IF (xClose) AND (NOT i_xClsLS) THEN
	q_xClose_A := TRUE;
	q_xClose_B := TRUE;
	q_xClose_C := TRUE;
END_IF
IF(CloseTimer.Q) OR (i_xClsLS) THEN
	q_xClose_A := FALSE;
	q_xClose_B := FALSE;
	q_xClose_C := FALSE;
	xClose := FALSE;
	iq_stValve.pv_xOPN_SW := FALSE;
END_IF

IF(OpenTimer.Q) AND (i_xOpnLS) THEN
	iq_stValve.q_xOPN_DO :=  FALSE;
	iq_stValve.pv_xOPN_SW := FALSE;
	xOpen:=FALSE;
END_IF

(* Neighboring Valves Interlock bit is reset When the Vacuum event error is reset and the Shutter is opened *)
IF (NOT i_xTrigger) AND (NOT iq_stValve.xERR_ExtFault) AND i_xOpnLS THEN
	q_xVAC_FAULT_OK := TRUE;
END_IF

(*OPN OK evaluation bit *)
iq_stValve.xOPN_OK := (NOT iq_stValve.xERR_ExtFault) AND NOT i_xTrigger;

(* If Epics Command to close the Valve, check if PMPS, otherwise Keep command set to open valve *)
// is there really a PMPS requirment.



(* When the valve  is open MPS is OK*)
q_xMPS_OK := (iq_stValve.eState=OPEN) AND NOT i_xTrigger AND i_xPress_OK;//gauge is connected


(* Override logic *)
(* Goal: give ability to override, but do so in a way that people won't forget it.
Solution: Override only after ten seconds of override, protect against blips,
when the valve permission goes true for more than ten seconds consistently, remove override
*)

tonDelOK(IN:=iq_stValve.xOPN_OK, PT:=tDelOK);
rtOK(CLK:=tonDelOK.Q);
IF rtOK.Q AND iq_stValve.pv_xOvrdOpn THEN 
	iq_stValve.pv_xOvrdOpn :=FALSE;
	//iq_stValve.pv_xOPN_SW := TRUE; //for seamless transition
END_IF

//Override timer
tonOvrd(IN:=iq_stValve.pv_xOvrdOpn, PT:=tOvrd);



///Check valve postion timout
IF NOT iq_stValve.i_xClsLS AND tCLStimeout.Q THEN 
	iq_stValve.bErrorPresent := TRUE;
ELSIF NOT iq_stValve.i_xOpnLS AND tOPNtimeout.Q THEN 
	iq_stValve.bErrorPresent := TRUE;
END_IF

(*Timers*)
CloseTimer ( IN:=xClose, PT:= TimDur, Q=>);
OpenTimer ( IN:=xOpen, PT:= OpenTimDur, Q=>);
tOPNtimeout(IN:= iq_stValve.q_xOPN_DO, PT := tTimeOutDuration );
tCLStimeout(IN:= NOT iq_stValve.q_xOPN_DO, PT := tTimeOutDuration);

(* Soft IO Mapping*)
IO();
// Alarm reset
//////////////////////////////////////
ACT_ResetAlarms();

ACTION ACT_ResetAlarms:
iq_stValve.xERR_DifPres R= i_xResetFault;

iq_stValve.bErrorPresent R= i_xResetFault;

IF NOT i_xTrigger  THEN
	iq_stValve.xERR_ExtFault R= i_xResetFault;
END_IF
END_ACTION

ACTION IO:
(*inputs*)
iq_stValve.i_xOpnLS := 	i_xOpnLS;
iq_stValve.i_xClsLS:=	i_xClsLS;
iq_stValve.xEXT_OK := i_xEXT_OK;
iq_stValve.xOverrideMode := i_xOverrideMode;
(*outputs*)
q_xOPN_DO:= iq_stValve.q_xOPN_DO;
q_xTrigger:=i_xTrigger;

//iq_stValve.pv_xOPN_SW:= i_xOPN_SW;

q_xVFS_Closed:= iq_stValve.i_xClsLS;
q_xVFS_Open:= iq_stValve.i_xOpnLS;
END_ACTION

END_FUNCTION_BLOCK

// POUs/Functions/Valves/FB_VGC
(* This function block implements basic functionality for Isolation Gate Valves*)
(* This function block interlock is as follows:
1. The valve can be opened when the difference between the pressures on both sides is
less than the maximum differential pressure.
2. This rule persists until the pressures on both sides are lower than the vacuum-setpoint.
3. Once at-vac, the valve will close if the pressure on either side rises above the setpoint.*)
(*This function block also implements PMPS and EPS interlocks, as well as Fast MPS trigger*)
FUNCTION_BLOCK FB_VGC
VAR_IN_OUT
	
END_VAR
VAR_INPUT
	(*Upstream Gauge, usually ion gauge*)
	i_stUSG	:	ST_VG;
	(*Downstream Gauge, usually ion gauge*)
	i_stDSG	:	ST_VG;
	{attribute 'pytmc' := '
    pv: Dis_DPIlk
	'}
	i_xDis_DPIlk : BOOL := FALSE;  (* Set to true when calling the function to disable the differential pressure interlock *)
	{attribute 'pytmc' := '
    pv: EPS_OK
	'}
	i_xEPS_OK:	BOOL	:= TRUE; (*External EPS interlock, Set to TRUE when no EPS interlock is required, otherwise set to correct interlock signal*)
	{attribute 'pytmc' := '
    pv: MPS_OK
	'}
	i_xPMPS_OK:	BOOL	; (*External MPS interlock, Set to TRUE when no PMPS interlock is required*)
		i_xExt_OK: BOOL; (*Other External Interlock, Set to True when no external interlock is required. If this Valve is neigboring a Fast Shutter this should be linked to the fast shutter xVAC_FAULT_OK*)
	i_xOverrideMode : BOOL; (*To be linked to global override bit. This Overrides Vacuum logic only, EPS, MPS and PMPS are still enforces*)
	// Reset fault
	{attribute 'pytmc' := '
    pv: FF_Reset
	'}
    i_xReset: BOOL;
END_VAR
VAR_OUTPUT
	{attribute 'pytmc' := '
    pv:
	'}
	iq_stValve : ST_VGC; (* All valve data and states will be in this struct*)
	
	{attribute 'pytmc' := '
    pv: MPS_FAULT_OK
	field: ZNAM MPS FAULT ;
	field: ONAM MPS OK ;
	'}
	xMPS_OK:	BOOL; (*MPS Fast OK, is set when the Valve is Open*)
END_VAR
VAR_IN_OUT
	io_fbFFHWO    :    FB_HardwareFFOutput;
END_VAR
VAR
	// PMPS
	fbFF    :    FB_FastFault :=(
        i_DevName := 'VGC',
        i_Desc := 'Fault occurs when the valve is not in open state',
        i_TypeCode := 16#1010);
	//g_FastFaultOutput1	:	FB_HardwareFFOutput;	

	{attribute 'instance-path'}
	{attribute 'noinit'}
	sPath: STRING;
	
	rDiffPressAllowed	:	REAL := 22.5; // Torr, Default value comes from Vat Valve Manual
	rDiffPress : REAL;
	set : BOOL;
    reset: BOOL;
	  
	xFirstPass	:	BOOL;
	fbFSInit		:	R_TRIG;
	
	tonDelOK : TON;
	rtOK	:	R_TRIG;
	tonOvrd	:	TON;
	
	tDelOK	:	TIME := T#60S;
	tOvrd	:	TIME := T#10s;
	
	
	(* Timeouts*)
	tTimeOutDuration: TIME:= T#5S;
	tOPNtimeout: TON;
	tCLStimeout:TON;
	
	
	(*IO*)
	i_xOpnLS	AT%I*: BOOL;
	i_xClsLS	AT%I*: BOOL;
	q_xOPN_DO	AT%Q*: BOOL;
    
    // For logging
    fbLogger : FB_LogMessage := (eSubsystem:=E_SubSystem.VACUUM);
    ePrevState : E_VGC;
    tErrorPresent : R_TRIG;
    tAction : R_TRIG; // Primary action of this device (OPN_DO, PUMP_RUN, etc.)
    tOverrideActivated : R_TRIG;
	
END_VAR

(* Vacuum gate valve
A. Wallace
16-10-29

A gate valve isolates vacuum volumes. Ideally it can be opened when a system is vented
to allow for faster pumping, and will close when high vacuum is lost.

The following behavior is good for valves in something like a gas attenuator.
This function block does the following:
1. The valve can be opened when the difference between the pressures on both sides is
less than the maximum differential pressure.
2. This rule persists until the pressures on both sides are lower than the vacuum-setpoint.
3. Once at-vac, the valve will close if the pressure on either side rises above the setpoint.

Alternatively, the differential pressure interlock can be disabled so the valve may only be opened
if the pressure on both sides is lower than the at-vacuum-setpoint. You want this behavior if 
the valve is to be used in a UHV section.

Hysteresis is employed to ensure a smooth transition from vented/pumping down, to at-vac.

Finally, an override system is built in so you can bypass all the interlocking logic and 
get back online.
*)
(* 10/1/2018 Margaret Ghaly included EPS, PMPS Checkes and MPS trigger signals*)


fbFSInit( CLK := TRUE, Q => xFirstPass);
(*IO Mapping*)
ACT_IO();

(* On first PLC pass, put valve into vented state, which implies a closed valve *)
IF xFirstPass THEN
	iq_stValve.eVGC_State := Vented;
	iq_stValve.pv_xOPN_SW := FALSE;
END_IF


///Check valve postion
IF iq_stValve.i_xClsLS AND  iq_stValve.i_xOpnLS THEN
	iq_stValve.eState:=INVALID;
ELSIF NOT iq_stValve.i_xClsLS AND iq_stValve.i_xOpnLS AND iq_stValve.q_xOPN_DO THEN 
	iq_stValve.eState:=OPEN;
ELSIF iq_stValve.i_xClsLS AND NOT iq_stValve.i_xOpnLS AND NOT iq_stValve.q_xOPN_DO THEN 
	iq_stValve.eState:=CLOSED;
ELSIF NOT iq_stValve.i_xClsLS AND NOT iq_stValve.i_xOpnLS THEN 
	iq_stValve.eState:=MOVING;
ELSE
	iq_stValve.eState:=INVALID;
END_IF

// Update hysteresis
///////////////////////////////////////////////////
IF iq_stValve.rAT_VAC_SP_LAST <> iq_stValve.rAT_VAC_SP OR xFirstPass THEN
	iq_stValve.rAT_VAC_SP_LAST := iq_stValve.rAT_VAC_SP;
	iq_stValve.rAT_VAC_HYS := iq_stValve.rHYST_PERC * iq_stValve.rAT_VAC_SP;
END_IF

iq_stValve.rAT_VAC_HYS := LIMIT(0, iq_stValve.rAT_VAC_HYS, iq_stValve.rAT_VAC_SP);
IF iq_stValve.rAT_VAC_SP <> 0 THEN
	IF iq_stValve.rHYST_PERC <> (iq_stValve.rAT_VAC_HYS / iq_stValve.rAT_VAC_SP) THEN
		iq_stValve.rHYST_PERC := LIMIT(0, (iq_stValve.rAT_VAC_HYS / iq_stValve.rAT_VAC_SP) ,1);
	END_IF
END_IF
// Valve at vacuum check
///////////////////////////////////////////////////
	set := i_stUSG.rPRESS < iq_stValve.rAT_VAC_HYS AND i_stDSG.rPRESS < iq_stValve.rAT_VAC_HYS AND i_stUSG.xPRESS_OK AND i_stDSG.xPRESS_OK;
 	iq_stValve.xAT_VAC S= set;
	reset := i_stUSG.rPRESS > iq_stValve.rAT_VAC_SP OR i_stDSG.rPRESS > iq_stValve.rAT_VAC_SP OR NOT i_stUSG.xPRESS_OK OR NOT i_stDSG.xPRESS_OK;
	iq_stValve.xAT_VAC R= reset;
	
// Differential pressure check
///////////////////////////////////////////////////
	(* Calc the differential pressure across the valve *)
	rDiffPress := ABS(i_stUSG.rPRESS - i_stDSG.rPRESS);
	
	(* As long as the differential pressure is less than 30mbar, the valve is allowed to open *)
	IF rDiffPress <= rDiffPressAllowed AND i_stUSG.xPRESS_OK AND i_stDSG.xPRESS_OK THEN
		iq_stValve.xDP_OK := TRUE;
	ELSE
		iq_stValve.xDP_OK	:= FALSE;
		(* If the differential pressure is exceeded, even when the valve is open,
		the state is unexpected and triggers a fault, because it suggests that something
		is wrong with the valve, or gauges or mapping or there is a major leak on one side.*)
		iq_stValve.eVGC_State := ERR_DiffPress;
        iq_stValve.xERR_DifPres := TRUE;
	END_IF

// Valve state
///////////////////////////////////////////////////
CASE iq_stValve.eVGC_State OF
	Vented: (* The Vented state is used during pump down *)
        //Log new state
        IF ePrevState <> iq_stValve.eVGC_State THEN
            fbLogger(sMsg:='Vented', eSevr:=TcEventSeverity.Info);
            ePrevState := iq_stValve.eVGC_State;
		END_IF
        
		(* Assuming the pump down went well, we are now at vacuum on both sides,
		so we move to the vacuum state, otherwise remain in the vented state *)
		IF iq_stValve.xAT_VAC AND (NOT (iq_stValve.xERR_DifPres)) AND NOT (NOT (iq_stValve.xERR_SP)) and NOT (NOT (iq_stValve.xERR_ExtFault))THEN
		    iq_stValve.eVGC_State := AtVacuum;
		ELSE
		    iq_stValve.eVGC_State := Vented;
		END_IF
	
	AtVacuum:
        //Log new state
        IF ePrevState <> iq_stValve.eVGC_State THEN
            fbLogger(sMsg:='Vacuum setpoint satisfied', eSevr:=TcEventSeverity.Info);
            ePrevState := iq_stValve.eVGC_State;
		END_IF
        
		IF iq_stValve.xAT_VAC THEN
		(* If both pressure setpoints are made,
		then enable the differential pressure interlock, regardless of the valve state
		assuming we're using some kind of ion gauge where a pressure setpoint cannot be higher than 1E-4 T *)
		iq_stValve.eVGC_State := AtVacuum;
				
		ELSE
		
			(* If the valve is open (or in an unknown state) and either gauge is not at it's vacuum setpoint,
			we have a loss of vacuum error *)
			IF (iq_stValve.i_xOpnLS OR (NOT iq_stValve.i_xOpnLS AND NOT iq_stValve.i_xClsLS)) THEN
				iq_stValve.eVGC_State := ERR_LostVac;
				iq_stValve.xERR_SP := TRUE; //TAW changed this to the ERR_SP bool because I think that's what it was intended to be?
		
			(* Alternatively, if the valve is already closed and we lose pressure on one side,
			it was probably intentional venting, so we calmly move back to venting mode, and
			disable the differential pressure interlock *) //?? 
			ELSIF iq_stValve.i_xClsLS THEN
				iq_stValve.eVGC_State := Vented;
			END_IF
		
		END_IF
	
	ERR_DiffPress:
        //Log new state
        IF ePrevState <> iq_stValve.eVGC_State THEN
            fbLogger(sMsg:='Potential accidental vent.', eSevr:=TcEventSeverity.Critical);
            ePrevState := iq_stValve.eVGC_State;
		END_IF
        
		IF NOT (iq_stValve.xERR_DifPres) THEN
			iq_stValve.eVGC_State := Vented;
		END_IF
		
	
	ERR_LostVac:
        //Log new state
        IF ePrevState <> iq_stValve.eVGC_State THEN
            fbLogger(sMsg:='Unexpected loss of vacuum while valve was open.', eSevr:=TcEventSeverity.Critical);
            ePrevState := iq_stValve.eVGC_State;
		END_IF
		IF NOT (iq_stValve.xERR_SP) THEN
			iq_stValve.eVGC_State := Vented;
		END_IF
		
	ERR_ExtFault:
        //Log new state
        IF ePrevState <> iq_stValve.eVGC_State THEN
            fbLogger(sMsg:='Lost external interlock while valve was open.', eSevr:=TcEventSeverity.Critical);
            ePrevState := iq_stValve.eVGC_State;
		END_IF
		IF NOT (iq_stValve.xERR_ExtFault) AND (NOT i_xExt_OK) THEN
			iq_stValve.eVGC_State := Vented;
		END_IF
END_CASE

IF (NOT i_xExt_OK) THEN
	iq_stValve.eVGC_State := ERR_ExtFault;
	iq_stValve.xERR_ExtFault := TRUE;
END_IF

// Interlock evaluation - with bypass for DP ILK bypass
///////////////////////////////////////////////
IF i_xDis_DPIlk THEN
	iq_stValve.xOPN_OK := iq_stValve.xEXT_OK; // AND iq_stValve.xDP_OK ;
ELSE
	iq_stValve.xOPN_OK := iq_stValve.xEXT_OK AND iq_stValve.xAT_VAC;
END_IF


(* Valve operation *)

(* Override logic *)
(* Goal: give ability to override, but do so in a way that people won't forget it.
Solution: Override only after ten seconds of override, protect against blips,
when the valve permission goes true for more than ten seconds consistently, remove override
*)

tonDelOK(IN:=iq_stValve.xOPN_OK, PT:=tDelOK);
rtOK(CLK:=tonDelOK.Q);
IF rtOK.Q AND iq_stValve.pv_xOvrdOpn THEN 
	iq_stValve.pv_xOvrdOpn :=FALSE;
	iq_stValve.pv_xOPN_SW := TRUE; //for seamless transition
    
    //Log
    fbLogger(sMsg:='Override expired', eSevr:=TcEventSeverity.Warning);
    
END_IF

//Override timer
tonOvrd(IN:=iq_stValve.pv_xOvrdOpn, PT:=tOvrd);

(* If Epics Command to close the Valve, check if PMPS and EPS are ok, otherwise Keep command set to open valve *)
IF NOT(iq_stValve.pv_xOPN_SW) AND ((NOT i_xPMPS_OK) OR (NOT i_xEPS_OK)) THEN
	iq_stValve.pv_xOPN_SW := TRUE; // plc to only reset never to set this signal
END_IF
(* Reset the EPICS command to open the valve if the interlock is lost *) 
(* based on EPS ok state, EPS overrides OPN_OK*)
IF NOT iq_stValve.xOPN_OK THEN
	IF i_xEPS_OK THEN iq_stValve.pv_xOPN_SW := FALSE; iq_stValve.sErrorMessage := 'ILK Active';
	ELSE iq_stValve.pv_xOPN_SW := TRUE;		// plc to only reset never to set this signal
	END_IF
END_IF

(* Here's where the valve opens *)
iq_stValve.q_xOPN_DO := (iq_stValve.pv_xOPN_SW AND iq_stValve.xOPN_OK) OR (tonOvrd.Q AND i_xOverrideMode);

(* When the valve  is open MPS is OK*)
xMPS_OK := (iq_stValve.eState=OPEN);//iq_stValve.i_xOpnLS; 

///Check valve moving postion timout
IF NOT iq_stValve.i_xClsLS AND tCLStimeout.Q THEN 
	iq_stValve.bErrorPresent := TRUE;
	iq_stValve.sErrorMessage := ': Close Timeout';
ELSIF NOT iq_stValve.i_xOpnLS AND tOPNtimeout.Q THEN 
	iq_stValve.bErrorPresent := TRUE; 
	iq_stValve.sErrorMessage := ': Open Timeout';
END_IF
IF (iq_stValve.eState=INVALID) THEN
	iq_stValve.bErrorPresent := TRUE; 
	iq_stValve.sErrorMessage := CONCAT(sPath,': Invalid Valve Position');
END_IF


(*Timers*)
tOPNtimeout(IN:= iq_stValve.q_xOPN_DO, PT := tTimeOutDuration );
tCLStimeout(IN:= NOT iq_stValve.q_xOPN_DO, PT := tTimeOutDuration);

// Log valve timeouts
tErrorPresent(CLK:=iq_stValve.bErrorPresent);
IF tErrorPresent.Q THEN fbLogger(sMsg:=iq_stValve.sErrorMessage, eSevr:=TcEventSeverity.Warning); END_IF

// Log valve open
tAction(CLK:= iq_stValve.q_xOPN_DO);
IF tAction.Q THEN fbLogger(sMsg:='Valve commanded open', eSevr:=TcEventSeverity.Info); END_IF

// Log override mode enabled
tOverrideActivated(CLK:= (tonOvrd.Q AND i_xOverrideMode));
IF tOverrideActivated.Q THEN fbLogger(sMsg:='Valve override mode activated', eSevr:=TcEventSeverity.Warning); END_IF

// Alarm reset
//////////////////////////////////////
ACT_ResetAlarms();

(*IO Mapping*)
ACT_IO();

(*FAST FAULT*)
fbFF(i_xOK := xMPS_OK,
    i_xReset := i_xReset,
    io_fbFFHWO := io_fbFFHWO);

ACTION ACT_IO:
(*inputs*)
iq_stValve.i_xOpnLS := 	i_xOpnLS;
iq_stValve.i_xClsLS:=	i_xClsLS;
iq_stValve.xEXT_OK := i_xEXT_OK;
iq_stValve.xOverrideMode := i_xOverrideMode;
(*outputs*)
q_xOPN_DO:= iq_stValve.q_xOPN_DO;
END_ACTION

ACTION ACT_ResetAlarms:
iq_stValve.xERR_DifPres R= iq_stValve.pv_xAlmRst;
iq_stValve.xERR_SP R= iq_stValve.pv_xAlmRst;
iq_stValve.bErrorPresent R= iq_stValve.pv_xAlmRst;

IF ( iq_stValve.pv_xAlmRst) THEN
	iq_stValve.sErrorMessage :='';
END_IF
END_ACTION

METHOD PUBLIC M_IsClosed : BOOL
VAR_INPUT
END_VAR
M_IsClosed := (This^.iq_stValve.eState = E_ValvePositionState.CLOSED);
END_METHOD

METHOD PUBLIC M_IsOpen : BOOL
VAR_INPUT
END_VAR
M_IsOpen := (This^.iq_stValve.eState = E_ValvePositionState.OPEN);
END_METHOD

// Use this Methode to Open or close the valve by setting the OPN_SW to the input value.
METHOD PUBLIC M_Set_OPN_SW : BOOL
VAR_INPUT
		value:BOOL;
END_VAR
This^.iq_stValve.pv_xOPN_SW := value;
END_METHOD

END_FUNCTION_BLOCK

// POUs/Functions/Valves/FB_VGC_AP
(* This function block implements basic functionality for Isolation Gate Valves with Appertures*)
(* This function block interlock is as follows:
1. The valve can be opened when the difference between the pressures on both sides is
less than the maximum differential pressure.
2. This rule persists until the pressures on both sides are lower than the vacuum-setpoint.
3. Once at-vac, the valve will close if the pressure on either side rises above the setpoint.*)
(*This function block also implements PMPS and EPS interlocks, as well as Fast MPS trigger*)
(* MPS is triggered differently than the VGC *)
FUNCTION_BLOCK FB_VGC_AP
VAR_IN_OUT
	
END_VAR
VAR_INPUT
	(*Upstream Gauge, usually ion gauge*)
	i_stUSG	:	ST_VG;
	(*Downstream Gauge, usually ion gauge*)
	i_stDSG	:	ST_VG;
	{attribute 'pytmc' := '
    pv: Dis_DPIlk
	'}
	i_xDis_DPIlk : BOOL := FALSE;  (* Set to true when calling the function to disable the differential pressure interlock *)
	{attribute 'pytmc' := '
    pv: EPS_OK
	'}
	i_xEPS_OK:	BOOL	:= TRUE; (*External EPS interlock, Set to TRUE when no EPS interlock is required, otherwise set to correct interlock signal*)
	{attribute 'pytmc' := '
    pv: MPS_OK
	'}
	i_xPMPS_OK:	BOOL	; (*External MPS interlock, Set to TRUE when no PMPS interlock is required*)
	i_xExt_OK: BOOL; (*Other External Interlock, Set to True when no external interlock is required. If this Valve is neigboring a Fast Shutter this should be linked to the fast shutter xVAC_FAULT_OK*)
	i_xOverrideMode : BOOL; (*To be linked to global override bit. This Overrides Vacuum logic only, EPS, MPS and PMPS are still enforces*)
	// Reset fault
	{attribute 'pytmc' := '
    pv: FF_Reset
	'}
    i_xReset: BOOL;
END_VAR
VAR_OUTPUT
	{attribute 'pytmc' := '
    pv:
	'}
	iq_stValve : ST_VGC; (* All valve data and states will be in this struct*)
	
	{attribute 'pytmc' := '
    pv: MPS_FAULT_OK
	'}
	xMPS_OK:	BOOL; (*MPS Fast OK, is set when the Valve is Open*)
END_VAR
VAR_IN_OUT
	io_fbFFHWO    :    FB_HardwareFFOutput;
END_VAR
VAR
	// PMPS
	fbFF    :    FB_FastFault :=(
        i_DevName := 'VGC',
        i_Desc := 'Fault occurs when the valve is not in open state',
        i_TypeCode := 16#1010);
	//g_FastFaultOutput1	:	FB_HardwareFFOutput;	

	{attribute 'instance-path'}
	{attribute 'noinit'}
	sPath: STRING;
	
	rDiffPressAllowed	:	REAL := 22.5; // Torr, Default value comes from Vat Valve Manual
	rDiffPress : REAL;
	set : BOOL;
    reset: BOOL;
	  
	xFirstPass	:	BOOL;
	fbFSInit		:	R_TRIG;
	
	tonDelOK : TON;
	rtOK	:	R_TRIG;
	tonOvrd	:	TON;
	
	tDelOK	:	TIME := T#60S;
	tOvrd	:	TIME := T#10s;
	
	
	(* Timeouts*)
	tTimeOutDuration: TIME:= T#5S;
	tOPNtimeout: TON;
	tCLStimeout:TON;
	
	
	(*IO*)
	i_xOpnLS	AT%I*: BOOL;
	i_xClsLS	AT%I*: BOOL;
	q_xOPN_DO	AT%Q*: BOOL;
	
END_VAR

(* Vacuum gate valve
A. Wallace
16-10-29

A gate valve isolates vacuum volumes. Ideally it can be opened when a system is vented
to allow for faster pumping, and will close when high vacuum is lost.

The following behavior is good for valves in something like a gas attenuator.
This function block does the following:
1. The valve can be opened when the difference between the pressures on both sides is
less than the maximum differential pressure.
2. This rule persists until the pressures on both sides are lower than the vacuum-setpoint.
3. Once at-vac, the valve will close if the pressure on either side rises above the setpoint.

Alternatively, the differential pressure interlock can be disabled so the valve may only be opened
if the pressure on both sides is lower than the at-vacuum-setpoint. You want this behavior if 
the valve is to be used in a UHV section.

Hysteresis is employed to ensure a smooth transition from vented/pumping down, to at-vac.

Finally, an override system is built in so you can bypass all the interlocking logic and 
get back online.
*)
(* 10/1/2018 Margaret Ghaly included EPS, PMPS Checkes and MPS trigger signals*)


fbFSInit( CLK := TRUE, Q => xFirstPass);
(*IO Mapping*)
ACT_IO();

(* On first PLC pass, put valve into vented state, which implies a closed valve *)
IF xFirstPass THEN
	iq_stValve.eVGC_State := Vented;
	iq_stValve.pv_xOPN_SW := FALSE;
END_IF


///Check valve postion
IF iq_stValve.i_xClsLS AND  iq_stValve.i_xOpnLS THEN
	iq_stValve.eState:=INVALID;
ELSIF NOT iq_stValve.i_xClsLS AND iq_stValve.i_xOpnLS AND iq_stValve.q_xOPN_DO THEN 
	iq_stValve.eState:=OPEN;
ELSIF iq_stValve.i_xClsLS AND NOT iq_stValve.i_xOpnLS AND NOT iq_stValve.q_xOPN_DO THEN 
	iq_stValve.eState:=CLOSED;
ELSIF NOT iq_stValve.i_xClsLS AND NOT iq_stValve.i_xOpnLS THEN 
	iq_stValve.eState:=MOVING;
ELSE
	iq_stValve.eState:=INVALID;
END_IF

// Update hysteresis
///////////////////////////////////////////////////
IF iq_stValve.rAT_VAC_SP_LAST <> iq_stValve.rAT_VAC_SP OR xFirstPass THEN
	iq_stValve.rAT_VAC_SP_LAST := iq_stValve.rAT_VAC_SP;
	iq_stValve.rAT_VAC_HYS := iq_stValve.rHYST_PERC * iq_stValve.rAT_VAC_SP;
END_IF

iq_stValve.rAT_VAC_HYS := LIMIT(0, iq_stValve.rAT_VAC_HYS, iq_stValve.rAT_VAC_SP);
IF iq_stValve.rAT_VAC_SP <> 0 THEN
	IF iq_stValve.rHYST_PERC <> (iq_stValve.rAT_VAC_HYS / iq_stValve.rAT_VAC_SP) THEN
		iq_stValve.rHYST_PERC := LIMIT(0, (iq_stValve.rAT_VAC_HYS / iq_stValve.rAT_VAC_SP) ,1);
	END_IF
END_IF
// Valve at vacuum check
///////////////////////////////////////////////////
	set := i_stUSG.rPRESS < iq_stValve.rAT_VAC_HYS AND i_stDSG.rPRESS < iq_stValve.rAT_VAC_HYS AND i_stUSG.xPRESS_OK AND i_stDSG.xPRESS_OK;
 	iq_stValve.xAT_VAC S= set;
	reset := i_stUSG.rPRESS > iq_stValve.rAT_VAC_SP OR i_stDSG.rPRESS > iq_stValve.rAT_VAC_SP OR NOT i_stUSG.xPRESS_OK OR NOT i_stDSG.xPRESS_OK;
	iq_stValve.xAT_VAC R= reset;
	
// Differential pressure check
///////////////////////////////////////////////////
	(* Calc the differential pressure across the valve *)
	rDiffPress := ABS(i_stUSG.rPRESS - i_stDSG.rPRESS);
	
	(* As long as the differential pressure is less than 30mbar, the valve is allowed to open *)
	IF rDiffPress <= rDiffPressAllowed AND i_stUSG.xPRESS_OK AND i_stDSG.xPRESS_OK THEN
		iq_stValve.xDP_OK := TRUE;
	ELSE
		iq_stValve.xDP_OK	:= FALSE;
		(* If the differential pressure is exceeded, even when the valve is open,
		the state is unexpected and triggers a fault, because it suggests that something
		is wrong with the valve, or gauges or mapping or there is a major leak on one side.*)
		iq_stValve.eVGC_State := ERR_DiffPress;
	END_IF

// Valve state
///////////////////////////////////////////////////
CASE iq_stValve.eVGC_State OF
	Vented: (* The Vented state is used during pump down *)
		(* Assuming the pump down went well, we are now at vacuum on both sides,
		so we move to the vacuum state, otherwise remain in the vented state *)
		IF iq_stValve.xAT_VAC THEN
		iq_stValve.eVGC_State := AtVacuum;
		ELSE
		iq_stValve.eVGC_State := Vented;
		END_IF
	
	AtVacuum:
		IF iq_stValve.xAT_VAC THEN
		(* If both pressure setpoints are made,
		then enable the differential pressure interlock, regardless of the valve state
		assuming we're using some kind of ion gauge where a pressure setpoint cannot be higher than 1E-4 T *)
		iq_stValve.eVGC_State := AtVacuum;
		ELSE
		
			(* If the valve is open (or in an unknown state) and either gauge is not at it's vacuum setpoint,
			we have a loss of vacuum error *)
			IF (iq_stValve.i_xOpnLS OR (NOT iq_stValve.i_xOpnLS AND NOT iq_stValve.i_xClsLS)) THEN
			iq_stValve.eVGC_State := ERR_LostVac;
		
			(* Alternatively, if the valve is already closed and we lose pressure on one side,
			it was probably intentional venting, so we calmly move back to venting mode, and
			disable the differential pressure interlock *) //?? 
			ELSIF iq_stValve.i_xClsLS THEN
			iq_stValve.eVGC_State := Vented;
			END_IF
		
		END_IF
	
	ERR_DiffPress:
		iq_stValve.eVGC_State := Vented;
		iq_stValve.xERR_DifPres := TRUE;
	
	ERR_LostVac:
		iq_stValve.eVGC_State := Vented;
		iq_stValve.xERR_SP := TRUE;
	
	END_CASE




// Interlock evaluation - with bypass for DP ILK bypass
///////////////////////////////////////////////
IF i_xDis_DPIlk THEN
	iq_stValve.xOPN_OK := iq_stValve.xEXT_OK; // AND iq_stValve.xDP_OK ;
ELSE
	iq_stValve.xOPN_OK := iq_stValve.xEXT_OK AND iq_stValve.xAT_VAC;
END_IF


(* Valve operation *)

(* Override logic *)
(* Goal: give ability to override, but do so in a way that people won't forget it.
Solution: Override only after ten seconds of override, protect against blips,
when the valve permission goes true for more than ten seconds consistently, remove override
*)

tonDelOK(IN:=iq_stValve.xOPN_OK, PT:=tDelOK);
rtOK(CLK:=tonDelOK.Q);
IF rtOK.Q AND iq_stValve.pv_xOvrdOpn THEN 
	iq_stValve.pv_xOvrdOpn :=FALSE;
	iq_stValve.pv_xOPN_SW := TRUE; //for seamless transition
END_IF

//Override timer
tonOvrd(IN:=iq_stValve.pv_xOvrdOpn, PT:=tOvrd);

(* If Epics Command to close the Valve, check if PMPS and EPS are ok, otherwise Keep command set to open valve *)
IF NOT(iq_stValve.pv_xOPN_SW) AND ((NOT i_xPMPS_OK) OR (NOT i_xEPS_OK)) THEN
	iq_stValve.pv_xOPN_SW := TRUE; // plc to only reset never to set this signal
END_IF
(* Reset the EPICS command to open the valve if the interlock is lost *) 
(* based on EPS ok state, EPS overrides OPN_OK*)
IF NOT iq_stValve.xOPN_OK THEN
	IF i_xEPS_OK THEN iq_stValve.pv_xOPN_SW := FALSE; iq_stValve.sErrorMessage := 'ILK Active';
	ELSE iq_stValve.pv_xOPN_SW := TRUE;		// plc to only reset never to set this signal
	END_IF
END_IF

(* Here's where the valve opens *)
iq_stValve.q_xOPN_DO := (iq_stValve.pv_xOPN_SW AND iq_stValve.xOPN_OK) OR (tonOvrd.Q AND i_xOverrideMode);

(* When the valve  is open MPS is OK*)
xMPS_OK := (iq_stValve.eState=OPEN) OR (iq_stValve.eState=CLOSED);//iq_stValve.i_xOpnLS; 

///Check valve moving postion timout
IF NOT iq_stValve.i_xClsLS AND tCLStimeout.Q THEN 
	iq_stValve.bErrorPresent := TRUE;
	iq_stValve.sErrorMessage := ': Close Timeout';
ELSIF NOT iq_stValve.i_xOpnLS AND tOPNtimeout.Q THEN 
	iq_stValve.bErrorPresent := TRUE; 
	iq_stValve.sErrorMessage := ': Open Timeout';
END_IF
IF (iq_stValve.eState=INVALID) THEN
	iq_stValve.bErrorPresent := TRUE; 
	iq_stValve.sErrorMessage := CONCAT(sPath,': Invalid Valve Position');
END_IF
(*Timers*)
tOPNtimeout(IN:= iq_stValve.q_xOPN_DO, PT := tTimeOutDuration );
tCLStimeout(IN:= NOT iq_stValve.q_xOPN_DO, PT := tTimeOutDuration);


// Alarm reset
//////////////////////////////////////
ACT_ResetAlarms();

(*IO Mapping*)
ACT_IO();

(*FAST FAULT*)
fbFF(i_xOK := xMPS_OK,
    i_xReset := i_xReset,
    io_fbFFHWO := io_fbFFHWO);

ACTION ACT_IO:
(*inputs*)
iq_stValve.i_xOpnLS := 	i_xOpnLS;
iq_stValve.i_xClsLS:=	i_xClsLS;
iq_stValve.xEXT_OK := i_xEXT_OK;
iq_stValve.xOverrideMode := i_xOverrideMode;
(*outputs*)
q_xOPN_DO:= iq_stValve.q_xOPN_DO;
END_ACTION

ACTION ACT_ResetAlarms:
iq_stValve.xERR_DifPres R= iq_stValve.pv_xAlmRst;
iq_stValve.xERR_SP R= iq_stValve.pv_xAlmRst;
iq_stValve.bErrorPresent R= iq_stValve.pv_xAlmRst;

IF ( iq_stValve.pv_xAlmRst) THEN
	iq_stValve.sErrorMessage :='';
END_IF
END_ACTION

METHOD PUBLIC M_IsClosed : BOOL
VAR_INPUT
END_VAR
M_IsClosed := (This^.iq_stValve.eState = E_ValvePositionState.CLOSED);
END_METHOD

METHOD PUBLIC M_IsOpen : BOOL
VAR_INPUT
END_VAR
M_IsOpen := (This^.iq_stValve.eState = E_ValvePositionState.OPEN);
END_METHOD

// Use this Methode to Open or close the valve by setting the OPN_SW to the input value.
METHOD PUBLIC M_Set_OPN_SW : BOOL
VAR_INPUT
		value:BOOL;
END_VAR
This^.iq_stValve.pv_xOPN_SW := value;
END_METHOD

END_FUNCTION_BLOCK

// POUs/Functions/Valves/FB_VGC_EBD
(* This function block is similar to the FB_VGC, except it has 2 outputs to actuate the Valve*)
(* This function block implements basic functionality for Isolation Gate Valves*)
(* This function block interlock is as follows:
1. The valve can be opened when the difference between the pressures on both sides is
less than the maximum differential pressure.
2. This rule persists until the pressures on both sides are lower than the vacuum-setpoint.
3. Once at-vac, the valve will close if the pressure on either side rises above the setpoint.*)
(*This function block also implements PMPS and EPS interlocks, as well as Fast MPS trigger*)
FUNCTION_BLOCK FB_VGC_EBD
VAR_IN_OUT
	
END_VAR
VAR_INPUT
	(*Upstream Gauge, usually ion gauge*)
	i_stUSG	:	ST_VG;
	(*Downstream Gauge, usually ion gauge*)
	i_stDSG	:	ST_VG;
	{attribute 'pytmc' := '
    pv: Dis_DPIlk
	'}
	i_xDis_DPIlk : BOOL := FALSE;  (* Set to true when calling the function to disable the differential pressure interlock *)
	{attribute 'pytmc' := '
    pv: EPS_OK
	'}
	i_xEPS_OK:	BOOL	:= TRUE; (*External EPS interlock, Set to TRUE when no EPS interlock is required, otherwise set to correct interlock signal*)
	{attribute 'pytmc' := '
    pv: MPS_OK
	'}
	i_xPMPS_OK:	BOOL	; (*External MPS interlock, Set to TRUE when no PMPS interlock is required*)
	i_xExt_OK: BOOL; (*Other External Interlock, Set to True when no external interlock is required*)
	i_xOverrideMode : BOOL; (*To be linked to global override bit. This Overrides Vacuum logic only, EPS, MPS and PMPS are still enforces*)
	// Reset fault
	{attribute 'pytmc' := '
    pv: FF_Reset
	'}
    i_xReset: BOOL;
END_VAR
VAR_OUTPUT
	{attribute 'pytmc' := '
    pv:
	'}
	iq_stValve : ST_VGC; (* All valve data and states will be in this struct*)
	
	{attribute 'pytmc' := '
    pv: MPS_FAULT_OK
	field: ZNAM MPS FAULT ;
	field: ONAM MPS OK ;
	'}
	xMPS_OK:	BOOL; (*MPS Fast OK, is set when the Valve is Open*)
END_VAR
VAR_IN_OUT
	io_fbFFHWO    :    FB_HardwareFFOutput;
END_VAR
VAR
	// PMPS
	fbFF    :    FB_FastFault :=(
        i_DevName := 'VGC',
        i_Desc := 'Fault occurs when the valve is not in open state',
        i_TypeCode := 16#1010);
	{attribute 'instance-path'}
	{attribute 'noinit'}
	sPath: STRING;
	
	rDiffPressAllowed	:	REAL := 22.5; // Torr, Default value comes from Vat Valve Manual
	rDiffPress : REAL;
	set : BOOL;
    reset: BOOL;
	  
	xFirstPass	:	BOOL;
	fbFSInit		:	R_TRIG;
	
	tonDelOK : TON;
	rtOK	:	R_TRIG;
	tonOvrd	:	TON;
	
	tDelOK	:	TIME := T#60S;
	tOvrd	:	TIME := T#10s;
	
	
	(* Timeouts*)
	tTimeOutDuration: TIME:= T#5S;
	tOPNtimeout: TON;
	tCLStimeout:TON;
	
	
	(*IO*)
	i_xOpnLS	AT%I*: BOOL;
	i_xClsLS	AT%I*: BOOL;
	q_xOPN_DO	AT%Q*: BOOL;
	q_xOPN_DO_2	AT%Q*: BOOL;
	
END_VAR

(* Vacuum gate valve
A. Wallace
16-10-29

A gate valve isolates vacuum volumes. Ideally it can be opened when a system is vented
to allow for faster pumping, and will close when high vacuum is lost.

The following behavior is good for valves in something like a gas attenuator.
This function block does the following:
1. The valve can be opened when the difference between the pressures on both sides is
less than the maximum differential pressure.
2. This rule persists until the pressures on both sides are lower than the vacuum-setpoint.
3. Once at-vac, the valve will close if the pressure on either side rises above the setpoint.

Alternatively, the differential pressure interlock can be disabled so the valve may only be opened
if the pressure on both sides is lower than the at-vacuum-setpoint. You want this behavior if 
the valve is to be used in a UHV section.

Hysteresis is employed to ensure a smooth transition from vented/pumping down, to at-vac.

Finally, an override system is built in so you can bypass all the interlocking logic and 
get back online.
*)
(* 10/1/2018 Margaret Ghaly included EPS, PMPS Checkes and MPS trigger signals*)


fbFSInit( CLK := TRUE, Q => xFirstPass);
(*IO Mapping*)
ACT_IO();

(* On first PLC pass, put valve into vented state, which implies a closed valve *)
IF xFirstPass THEN
	iq_stValve.eVGC_State := Vented;
	iq_stValve.pv_xOPN_SW := FALSE;
END_IF


///Check valve postion
IF iq_stValve.i_xClsLS AND  iq_stValve.i_xOpnLS THEN
	iq_stValve.eState:=INVALID;
ELSIF NOT iq_stValve.i_xClsLS AND iq_stValve.i_xOpnLS AND iq_stValve.q_xOPN_DO THEN 
	iq_stValve.eState:=OPEN;
ELSIF iq_stValve.i_xClsLS AND NOT iq_stValve.i_xOpnLS AND NOT iq_stValve.q_xOPN_DO THEN 
	iq_stValve.eState:=CLOSED;
ELSIF NOT iq_stValve.i_xClsLS AND NOT iq_stValve.i_xOpnLS THEN 
	iq_stValve.eState:=MOVING;
ELSE
	iq_stValve.eState:=INVALID;
END_IF

// Update hysteresis
///////////////////////////////////////////////////
IF iq_stValve.rAT_VAC_SP_LAST <> iq_stValve.rAT_VAC_SP OR xFirstPass THEN
	iq_stValve.rAT_VAC_SP_LAST := iq_stValve.rAT_VAC_SP;
	iq_stValve.rAT_VAC_HYS := iq_stValve.rHYST_PERC * iq_stValve.rAT_VAC_SP;
END_IF

iq_stValve.rAT_VAC_HYS := LIMIT(0, iq_stValve.rAT_VAC_HYS, iq_stValve.rAT_VAC_SP);
IF iq_stValve.rAT_VAC_SP <> 0 THEN
	IF iq_stValve.rHYST_PERC <> (iq_stValve.rAT_VAC_HYS / iq_stValve.rAT_VAC_SP) THEN
		iq_stValve.rHYST_PERC := LIMIT(0, (iq_stValve.rAT_VAC_HYS / iq_stValve.rAT_VAC_SP) ,1);
	END_IF
END_IF
// Valve at vacuum check
///////////////////////////////////////////////////
	set := i_stUSG.rPRESS < iq_stValve.rAT_VAC_HYS AND i_stDSG.rPRESS < iq_stValve.rAT_VAC_HYS AND i_stUSG.xPRESS_OK AND i_stDSG.xPRESS_OK;
 	iq_stValve.xAT_VAC S= set;
	reset := i_stUSG.rPRESS > iq_stValve.rAT_VAC_SP OR i_stDSG.rPRESS > iq_stValve.rAT_VAC_SP OR NOT i_stUSG.xPRESS_OK OR NOT i_stDSG.xPRESS_OK;
	iq_stValve.xAT_VAC R= reset;
	
// Differential pressure check
///////////////////////////////////////////////////
	(* Calc the differential pressure across the valve *)
	rDiffPress := ABS(i_stUSG.rPRESS - i_stDSG.rPRESS);
	
	(* As long as the differential pressure is less than 30mbar, the valve is allowed to open *)
	IF rDiffPress <= rDiffPressAllowed AND i_stUSG.xPRESS_OK AND i_stDSG.xPRESS_OK THEN
		iq_stValve.xDP_OK := TRUE;
	ELSE
		iq_stValve.xDP_OK	:= FALSE;
		(* If the differential pressure is exceeded, even when the valve is open,
		the state is unexpected and triggers a fault, because it suggests that something
		is wrong with the valve, or gauges or mapping or there is a major leak on one side.*)
		iq_stValve.eVGC_State := ERR_DiffPress;
	END_IF

// Valve state
///////////////////////////////////////////////////
CASE iq_stValve.eVGC_State OF
	Vented: (* The Vented state is used during pump down *)
		(* Assuming the pump down went well, we are now at vacuum on both sides,
		so we move to the vacuum state, otherwise remain in the vented state *)
		IF iq_stValve.xAT_VAC THEN
		iq_stValve.eVGC_State := AtVacuum;
		ELSE
		iq_stValve.eVGC_State := Vented;
		END_IF
	
	AtVacuum:
		IF iq_stValve.xAT_VAC THEN
		(* If both pressure setpoints are made,
		then enable the differential pressure interlock, regardless of the valve state
		assuming we're using some kind of ion gauge where a pressure setpoint cannot be higher than 1E-4 T *)
		iq_stValve.eVGC_State := AtVacuum;
		ELSE
		
			(* If the valve is open (or in an unknown state) and either gauge is not at it's vacuum setpoint,
			we have a loss of vacuum error *)
			IF (iq_stValve.i_xOpnLS OR (NOT iq_stValve.i_xOpnLS AND NOT iq_stValve.i_xClsLS)) THEN
			iq_stValve.eVGC_State := ERR_LostVac;
		
			(* Alternatively, if the valve is already closed and we lose pressure on one side,
			it was probably intentional venting, so we calmly move back to venting mode, and
			disable the differential pressure interlock *) //?? 
			ELSIF iq_stValve.i_xClsLS THEN
			iq_stValve.eVGC_State := Vented;
			END_IF
		
		END_IF
	
	ERR_DiffPress:
		iq_stValve.eVGC_State := Vented;
		iq_stValve.xERR_DifPres := TRUE;
	
	ERR_LostVac:
		iq_stValve.eVGC_State := Vented;
		iq_stValve.xERR_SP := TRUE;
	
	END_CASE




// Interlock evaluation - with bypass for DP ILK bypass
///////////////////////////////////////////////
IF i_xDis_DPIlk THEN
	iq_stValve.xOPN_OK := iq_stValve.xEXT_OK; // AND iq_stValve.xDP_OK ;
ELSE
	iq_stValve.xOPN_OK := iq_stValve.xEXT_OK AND iq_stValve.xAT_VAC;
END_IF


(* Valve operation *)

(* Override logic *)
(* Goal: give ability to override, but do so in a way that people won't forget it.
Solution: Override only after ten seconds of override, protect against blips,
when the valve permission goes true for more than ten seconds consistently, remove override
*)

tonDelOK(IN:=iq_stValve.xOPN_OK, PT:=tDelOK);
rtOK(CLK:=tonDelOK.Q);
IF rtOK.Q AND iq_stValve.pv_xOvrdOpn THEN 
	iq_stValve.pv_xOvrdOpn :=FALSE;
	iq_stValve.pv_xOPN_SW := TRUE; //for seamless transition
END_IF

//Override timer
tonOvrd(IN:=iq_stValve.pv_xOvrdOpn, PT:=tOvrd);

(* If Epics Command to close the Valve, check if PMPS and EPS are ok, otherwise Keep command set to open valve *)
IF NOT(iq_stValve.pv_xOPN_SW) AND ((NOT i_xPMPS_OK) OR (NOT i_xEPS_OK)) THEN
	iq_stValve.pv_xOPN_SW := TRUE; // plc to only reset never to set this signal
END_IF
(* Reset the EPICS command to open the valve if the interlock is lost *) 
(* based on EPS ok state, EPS overrides OPN_OK*)
IF NOT iq_stValve.xOPN_OK THEN
	IF i_xEPS_OK THEN iq_stValve.pv_xOPN_SW := FALSE; iq_stValve.sErrorMessage := 'ILK Active';
	ELSE iq_stValve.pv_xOPN_SW := TRUE;		// plc to only reset never to set this signal
	END_IF
END_IF

(* Here's where the valve opens *)
iq_stValve.q_xOPN_DO := (iq_stValve.pv_xOPN_SW AND iq_stValve.xOPN_OK) OR (tonOvrd.Q AND i_xOverrideMode);

(* When the valve  is open MPS is OK*)
xMPS_OK := (iq_stValve.eState=OPEN);//iq_stValve.i_xOpnLS; 

///Check valve moving postion timout
IF NOT iq_stValve.i_xClsLS AND tCLStimeout.Q THEN 
	iq_stValve.bErrorPresent := TRUE;
	iq_stValve.sErrorMessage := ': Close Timeout';
ELSIF NOT iq_stValve.i_xOpnLS AND tOPNtimeout.Q THEN 
	iq_stValve.bErrorPresent := TRUE; 
	iq_stValve.sErrorMessage := ': Open Timeout';
END_IF
IF (iq_stValve.eState=INVALID) THEN
	iq_stValve.bErrorPresent := TRUE; 
	iq_stValve.sErrorMessage := CONCAT(sPath,': Invalid Valve Position');
END_IF
(*Timers*)
tOPNtimeout(IN:= iq_stValve.q_xOPN_DO, PT := tTimeOutDuration );
tCLStimeout(IN:= NOT iq_stValve.q_xOPN_DO, PT := tTimeOutDuration);


// Alarm reset
//////////////////////////////////////
ACT_ResetAlarms();

(*IO Mapping*)
ACT_IO();

(*FAST FAULT*)
fbFF(i_xOK := xMPS_OK,
    i_xReset := i_xReset,
    io_fbFFHWO := io_fbFFHWO);

ACTION ACT_IO:
(*inputs*)
iq_stValve.i_xOpnLS := 	i_xOpnLS;
iq_stValve.i_xClsLS:=	i_xClsLS;
iq_stValve.xEXT_OK := i_xEXT_OK;
iq_stValve.xOverrideMode := i_xOverrideMode;
(*outputs*)
q_xOPN_DO:= iq_stValve.q_xOPN_DO;
q_xOPN_DO_2:= iq_stValve.q_xOPN_DO;
END_ACTION

ACTION ACT_ResetAlarms:
iq_stValve.xERR_DifPres R= iq_stValve.pv_xAlmRst;
iq_stValve.xERR_SP R= iq_stValve.pv_xAlmRst;
iq_stValve.bErrorPresent R= iq_stValve.pv_xAlmRst;

IF ( iq_stValve.pv_xAlmRst) THEN
	iq_stValve.sErrorMessage :='';
END_IF
END_ACTION

METHOD PUBLIC M_IsClosed : BOOL
VAR_INPUT
END_VAR
M_IsClosed := (This^.iq_stValve.eState = E_ValvePositionState.CLOSED);
END_METHOD

METHOD PUBLIC M_IsOpen : BOOL
VAR_INPUT
END_VAR
M_IsOpen := (This^.iq_stValve.eState = E_ValvePositionState.OPEN);
END_METHOD

// Use this Methode to Open or close the valve by setting the OPN_SW to the input value.
METHOD PUBLIC M_Set_OPN_SW : BOOL
VAR_INPUT
		value:BOOL;
END_VAR
This^.iq_stValve.pv_xOPN_SW := value;
END_METHOD

END_FUNCTION_BLOCK

// POUs/Functions/Valves/FB_VRC
(* This Function Block Implements Basic Functionality for certain types of valves e.g Turbo Isolation valves, Apperture Valve.
This function block is interloked by an input (i_xExtILK_OK). This is so developers can interface with custom
interlocking logic outside this function block.*)
(* Note Interlock Logic is External *)
FUNCTION_BLOCK FB_VRC
VAR_IN_OUT
	
END_VAR
VAR_INPUT
	{attribute 'pytmc' := '
	pv: EXT_ILK_OK ;
	field: ZNAM NOT OK ;
	field: ONAM OK ;
	io: i ;
	'}
	i_xExtILK_OK : BOOL; //Connect to Interlock logic condition(e.g F_TURBO_VRC_ILK Function), otherwise, Set to True if the valve is not interlocked
	i_xOverrideMode : BOOL; (*To be linked to global override bit. This Overrides Vacuum logic only, EPS, MPS and PMPS are still enforces*)
END_VAR
VAR_OUTPUT
	{attribute 'pytmc' := '
    pv:
	'}
	iq_stValve : ST_VRC;
END_VAR
VAR
	{attribute 'instance-path'}
	{attribute 'noinit'}
	sPath: STRING;
	xFirstPass	:	BOOL;
	fbFSInit		:	R_TRIG;
	tonOvrd	:	TON;
	tonDelOK : TON;
	rtOK	:	R_TRIG;

	(*IO*)
	i_xOpnLS	AT%I*: BOOL;
	i_xClsLS	AT%I*: BOOL;
	q_xOPN_DO	AT%Q*: BOOL;
END_VAR


(* On first PLC pass, put valve into vented state, which implies a closed valve *)
fbFSInit( CLK := TRUE, Q => xFirstPass);
IF xFirstPass THEN
	iq_stValve.eVGC_State := Vented;
	iq_stValve.pv_xOPN_SW := FALSE;
END_IF




///Check valve postion
IF iq_stValve.i_xClsLS AND  iq_stValve.i_xOpnLS THEN
	iq_stValve.eState:=INVALID;
ELSIF NOT iq_stValve.i_xClsLS AND iq_stValve.i_xOpnLS AND iq_stValve.q_xOPN_DO THEN 
	iq_stValve.eState:=OPEN;
ELSIF iq_stValve.i_xClsLS AND NOT iq_stValve.i_xOpnLS AND NOT iq_stValve.q_xOPN_DO THEN 
	iq_stValve.eState:=CLOSED;
ELSIF NOT iq_stValve.i_xClsLS AND NOT iq_stValve.i_xOpnLS THEN 
	iq_stValve.eState:=MOVING;
ELSE
	iq_stValve.eState:=INVALID;
END_IF


(*evaluate Valve open external interlock*)
iq_stValve.xOPN_OK := i_xExtILK_OK;
IF NOT iq_stValve.xOPN_OK and NOT tonOvrd.Q THEN
	iq_stValve.pv_xOPN_SW := FALSE;
	iq_stValve.eVGC_State := ERR_ExtFault;
END_IF

IF (iq_stValve.q_xOPN_DO) AND (iq_stValve.xOPN_OK) THEN
	iq_stValve.eVGC_State := AtVacuum;
END_IF
	

(* Override logic *)
(* Goal: give ability to override, but do so in a way that people won't forget it.
Solution: Override only after ten seconds of override, protect against blips,
when the valve permission goes true for more than ten seconds consistently, remove override
*)

tonDelOK(IN:=iq_stValve.xOPN_OK, PT:=T#10S);
rtOK(CLK:=tonDelOK.Q);
IF rtOK.Q THEN iq_stValve.pv_xOvrdOpn :=FALSE; END_IF

//Override timer
tonOvrd(IN:=iq_stValve.pv_xOvrdOpn, PT:=T#10S);

(* Here's where the valve opens *)
iq_stValve.q_xOPN_DO := (iq_stValve.pv_xOPN_SW AND iq_stValve.xOPN_OK) OR (tonOvrd.Q AND i_xOverrideMode);

(*Soft IO Mapping*)
ACT_IO();

ACTION ACT_IO:
(*inputs*)
iq_stValve.i_xOpnLS := 	i_xOpnLS;
iq_stValve.i_xClsLS:=	i_xClsLS;
iq_stValve.xOverrideMode := i_xOverrideMode;
(*outputs*)
q_xOPN_DO:= iq_stValve.q_xOPN_DO;
END_ACTION

// Use this Methode to Open or close the valve by setting the OPN_SW to the input value.
METHOD PUBLIC M_Set_OPN_SW : BOOL
VAR_INPUT
	value:BOOL;
END_VAR
This^.iq_stValve.pv_xOPN_SW := value;
END_METHOD

END_FUNCTION_BLOCK

// POUs/Functions/Valves/FB_VRC_EBD
(* This function block is similar to the FB_VGC, except it has 2 outputs to actuate the Valve*)
(* This Function Block Implements Basic Functionality for certain types of valves e.g Turbo Isolation valves, Apperture Valve *)
(* Note Interlock Logic is External *)
FUNCTION_BLOCK FB_VRC_EBD
VAR_IN_OUT
	
END_VAR
VAR_INPUT
	i_xExtILK_OK : BOOL; //Connect to Interlock logic condition(e.g F_TURBO_VRC_ILK Function), otherwise, Set to True if the valve is not interlocked
	i_xOverrideMode : BOOL; (*To be linked to global override bit. This Overrides Vacuum logic only, EPS, MPS and PMPS are still enforces*)
END_VAR
VAR_OUTPUT
	{attribute 'pytmc' := '
    pv:
	'}
	iq_stValve : ST_VRC;
END_VAR
VAR

	tonOvrd	:	TON;
	tonDelOK : TON;
	rtOK	:	R_TRIG;

	(*IO*)
	i_xOpnLS	AT%I*: BOOL;
	i_xClsLS	AT%I*: BOOL;
	q_xOPN_DO	AT%Q*: BOOL;
	q_xOPN_DO_2	AT%Q*: BOOL;
END_VAR



///Check valve postion
IF NOT iq_stValve.i_xClsLS AND iq_stValve.i_xOpnLS THEN 
	iq_stValve.eState:=OPEN;
ELSIF iq_stValve.i_xClsLS AND NOT iq_stValve.i_xOpnLS THEN 
	iq_stValve.eState:=CLOSED;
ELSIF NOT iq_stValve.i_xClsLS AND NOT iq_stValve.i_xOpnLS THEN 
	iq_stValve.eState:=MOVING;
ELSE
	iq_stValve.eState:=INVALID;
END_IF

(*evaluate Valve open external interlock*)
iq_stValve.xOPN_OK := i_xExtILK_OK;
IF NOT iq_stValve.xOPN_OK and NOT tonOvrd.Q THEN
	iq_stValve.pv_xOPN_SW := FALSE;
END_IF

(* Override logic *)
(* Goal: give ability to override, but do so in a way that people won't forget it.
Solution: Override only after ten seconds of override, protect against blips,
when the valve permission goes true for more than ten seconds consistently, remove override
*)

tonDelOK(IN:=iq_stValve.xOPN_OK, PT:=T#10S);
rtOK(CLK:=tonDelOK.Q);
IF rtOK.Q THEN iq_stValve.pv_xOvrdOpn :=FALSE; END_IF

//Override timer
tonOvrd(IN:=iq_stValve.pv_xOvrdOpn, PT:=T#10S);

(* Here's where the valve opens *)
iq_stValve.q_xOPN_DO := (iq_stValve.pv_xOPN_SW AND iq_stValve.xOPN_OK) OR (tonOvrd.Q AND i_xOverrideMode);

(*Soft IO Mapping*)
ACT_IO();

ACTION ACT_IO:
(*inputs*)
iq_stValve.i_xOpnLS := 	i_xOpnLS;
iq_stValve.i_xClsLS:=	i_xClsLS;
iq_stValve.xOverrideMode := i_xOverrideMode;
(*outputs*)
q_xOPN_DO:= iq_stValve.q_xOPN_DO;
q_xOPN_DO_2:= iq_stValve.q_xOPN_DO;
END_ACTION

// Use this Methode to Open or close the valve by setting the OPN_SW to the input value.
METHOD PUBLIC M_Set_OPN_SW : BOOL
VAR_INPUT
	value:BOOL;
END_VAR
This^.iq_stValve.pv_xOPN_SW := value;
END_METHOD

END_FUNCTION_BLOCK

// POUs/Functions/Valves/FB_VRC_OK_CLS
(* This function block is different from the regular VRC in that CLOSING must be permitted. *)
FUNCTION_BLOCK FB_VRC_OK_CLS
VAR_IN_OUT
	iq_stValve : ST_VRC;
END_VAR
VAR_INPUT
	i_xOverrideMode : BOOL;
END_VAR
VAR_OUTPUT
END_VAR
VAR

tonOvrd	:	TON;
tonDelOK : TON;
rtOK	:	R_TRIG;

END_VAR

(* This function block is different from the regular VRC in that CLOSING must be permitted. *)
(* Implemented for the funky valve 04 on LAMP *)
IF NOT iq_stValve.xOPN_OK and NOT tonOvrd.Q THEN
iq_stValve.pv_xOPN_SW := FALSE;
END_IF

(* Override logic *)
(* Goal: give ability to override, but do so in a way that people won't forget it.
Solution: Override only after ten seconds of override, protect against blips,
when the valve permission goes true for more than ten seconds consistently, remove override
*)

tonDelOK(IN:=iq_stValve.xOPN_OK, PT:=T#10S);
rtOK(CLK:=tonDelOK.Q);
IF rtOK.Q THEN iq_stValve.pv_xOvrdOpn :=FALSE; END_IF

//Override timer
tonOvrd(IN:=iq_stValve.pv_xOvrdOpn, PT:=T#10S);

(* Here's where the valve opens *)
iq_stValve.q_xOPN_DO := NOT iq_stValve.xCLS_OK OR ((iq_stValve.pv_xOPN_SW AND iq_stValve.xOPN_OK) OR (tonOvrd.Q AND i_xOverrideMode));

END_FUNCTION_BLOCK
